
FUNCTION_BLOCK FB 1032
TITLE =A_3225_MXZ01MA FAN 1
//COPYRIGHT:     (C) 2009  BUHLER AG, CH-9240 UZWIL, SWITZERLAND
//
//PRODUCT:       WinCoS_BIW01_09
//
//TITLE:         FAN 1
//
//--------------------------------------------------------------------------------
//
//IDENT:         AUTHOR:             DEPT:                             DATE:
//
//P01_FB1032.1.0 K.Renz              CSB41                             09.Okt.2009
//               1st Release
//
//--------------------------------------------------------------------------------
//
//PURPOSE:
//
//MANUAL :
//
//RESTRICTIONS:
//
//--------------------------------------------------------------------------------
AUTHOR : KR
FAMILY : USW
VERSION : 0.0


VAR
  Ma : "GCS7_M_FB50_Data";	// Machine
  A_3225_KCU04 : "GCS7_E_DigInput";	// Mon1: DigInpCont
  A_3225_MXZ01_SM : "GCS7_E_DigInput";	// Mon2: DigInpCont
  Mon3 : "GCS7_E_DigInput";	// spare
  Mon4 : "GCS7_E_DigInput";	// spare
  Mon5 : "GCS7_E_DigInput";	// spare
  Mon6 : "GCS7_E_DigInput";	// spare
  A_3225_MXZ01 : "GCS7_E_Motor";	// Motor: Motor
END_VAR
BEGIN
NETWORK
TITLE =Call SSW

      UC    "GCS7_M_Motor6Mon";
END_FUNCTION_BLOCK


FUNCTION_BLOCK "G297M_Code"
TITLE =G297M FAN KILN 2
//COPYRIGHT:    (C) 2009  BUHLER AG, CH-9240 UZWIL, SWITZERLAND
//
//PRODUCT:      WinCoS_BIW01_09
//
//TITLE:        FAN KILN 2
//                Machine group control
//                Maschinengruppensteuerung
//
//--------------------------------------------------------------------------------
//
//IDENT:        AUTHOR:             DEPT:                              DATE:
//
//P01_FB397.1.0 K.Renz              CSB41                              09.Okt.2009
//             1st Release
//
//--------------------------------------------------------------------------------
//
//PURPOSE:
//
//MANUAL :
//
//RESTRICTIONS:
//
//--------------------------------------------------------------------------------
AUTHOR : KR
FAMILY : USW
VERSION : 9.9


VAR
  Gr : "GCS7_GrpCtrlSub";	//Standard interface to group
  InOutValue1 : DINT ;	//Data for user
  InOutValue2 : DINT ;	//Data for user
  OutWayConflict : BOOL ;	//Data for user
  OutSelectionOk : BOOL ;	//Data for user
  CmdNewValue : BOOL ;	//Data for user
  CmdNewJob : BOOL ;	//Data for user
  OutCodeOK : BOOL ;	//Data for user
  InEndOfJob : BOOL ;	//Data for user
  staWayOk : BOOL ;	//Data for user
  EdgeStartRelease : BOOL ;	//Data for user
  USW8 : BOOL ;	//Data for user
  USW9 : BOOL ;	//Data for user
  USW10 : BOOL ;	//Data for user
  USW11 : BOOL ;	//Data for user
  USW12 : BOOL ;	//Data for user
  USW13 : BOOL ;	//Data for user
  USW14 : BOOL ;	//Data for user
  USW15 : BOOL ;	//Data for user
  A_3225_KCU04AI1 : "GCS7_E_AnalogInput";	// AnaInp
  A_3225_KCU04AI2 : "GCS7_E_AnalogInput";	// AnaInp
  A_3225_BTE05 : "GCS7_E_AnalogInput";	// AnaInp
  A_3225_BTE06 : "GCS7_E_AnalogInput";	// AnaInp
  spare412 : ARRAY  [412 .. 445 ] OF BYTE ;
  A_3225_MXZ01MA : FB 1032;	// Motor+6DI
  A_3225_TSC01_AC : "GCS7_E_AnalogInput";	// AnaInp
  A_3225_TSC01_AF : "GCS7_E_AnalogInput";	// AnaInp
  A_3225_TSC01_AP : "GCS7_E_AnalogInput";	// AnaInp
  A_3225_TSC01_AT : "GCS7_E_AnalogInput";	// AnaInp
  A_3225_TSC01_COM : "SSA_SEW_MOVIDRIVE";	// FU_Siemens
  A_3226_KCU04AI1 : "GCS7_E_AnalogInput";	// AnaInp
  A_3226_KCU04AI2 : "GCS7_E_AnalogInput";	// AnaInp
  A_3226_BTE05 : "GCS7_E_AnalogInput";	// AnaInp
  A_3226_BTE06 : "GCS7_E_AnalogInput";	// AnaInp
  A_3226_MXZ01MA : FB 1033;	// Motor+6DI
  A_3226_TSC01_AC : "GCS7_E_AnalogInput";	// AnaInp
  A_3226_TSC01_AF : "GCS7_E_AnalogInput";	// AnaInp
  A_3226_TSC01_AP : "GCS7_E_AnalogInput";	// AnaInp
  A_3226_TSC01_AT : "GCS7_E_AnalogInput";	// AnaInp
  A_3226_TSC01_COM : "SSA_SEW_MOVIDRIVE";	// FU_Siemens
  A_3226_TSC01 : FB14;   // DigInpCont
END_VAR
VAR_TEMP
  tmpEnable : BOOL ;
  tmpFlag : BOOL ;
  tmpCmdNext : BOOL ;
  tmpLocal : BOOL ;
  tmpAspOk : BOOL ;
  tmpHWStop : BOOL ;
  tmpInstanzDBNo : INT ;
END_VAR
BEGIN
NETWORK
TITLE =



NETWORK
TITLE =Read command from group control
//Parameter
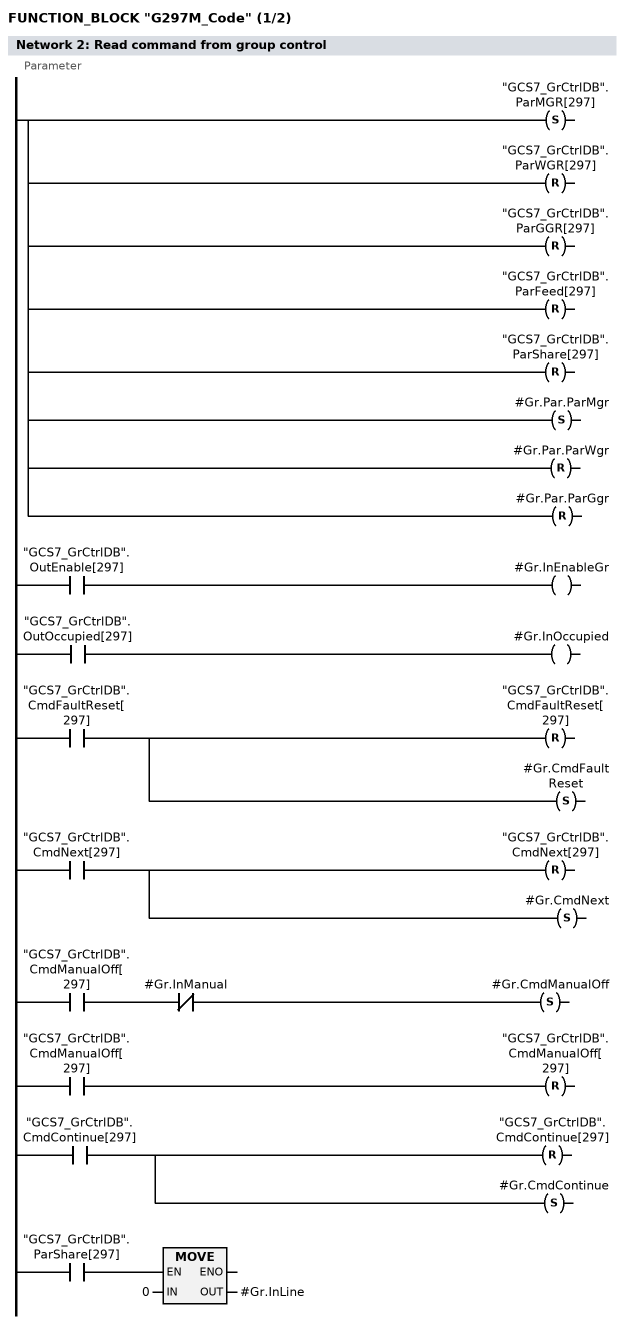
      SET   ;
      S     "GCS7_GrCtrlDB".ParMGR[297];
      R     "GCS7_GrCtrlDB".ParWGR[297];
      R     "GCS7_GrCtrlDB".ParGGR[297];
      R     "GCS7_GrCtrlDB".ParFeed[297];
      R     "GCS7_GrCtrlDB".ParShare[297];
      S     #Gr.Par.ParMgr;
      R     #Gr.Par.ParWgr;
      R     #Gr.Par.ParGgr;
//Command
      U     "GCS7_GrCtrlDB".OutEnable[297];
      =     #Gr.InEnableGr;
      U     "GCS7_GrCtrlDB".OutOccupied[297];
      =     #Gr.InOccupied;
      U     "GCS7_GrCtrlDB".CmdFaultReset[297];
      R     "GCS7_GrCtrlDB".CmdFaultReset[297];
      S     #Gr.CmdFaultReset;
      U     "GCS7_GrCtrlDB".CmdNext[297];
      R     "GCS7_GrCtrlDB".CmdNext[297];
      S     #Gr.CmdNext;

      U     "GCS7_GrCtrlDB".CmdManualOff[297];
      UN    #Gr.InManual;
      S     #Gr.CmdManualOff;
      U     "GCS7_GrCtrlDB".CmdManualOff[297];
      R     "GCS7_GrCtrlDB".CmdManualOff[297];

//      U     "GCS7_GrCtrlDB".CmdManualOff[297]
//      O     "GCS7_GrCtrlDB".OutOccupied[297]
//      R     "GCS7_GrCtrlDB".CmdManualOff[297]
//      S     #Gr.CmdManualOff

      U     "GCS7_GrCtrlDB".CmdContinue[297];
      R     "GCS7_GrCtrlDB".CmdContinue[297];
      S     #Gr.CmdContinue;
//Init Line Number
      U     "GCS7_GrCtrlDB".ParShare[297];
      SPBN  WE00;
      L     0;
      T     #Gr.InLine;
WE00: NOP   0;
NETWORK
TITLE =Call Methode Control
// 1. Handle Interface PCControl
// 2. Prepare mode --> ModePassive,ModeActive,ModeIdling
// 3. Reset global flags of the group
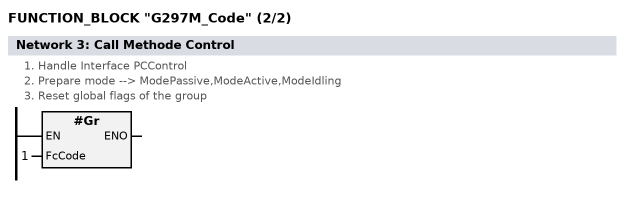
      CALL #Gr (
           FcCode                   := 1);
NETWORK
TITLE =Restart Idling Time

      L     #Gr.Par.ParIdling;
      L     2;
      >=I   ;
      SPB   IdTm;
      T     #Gr.Par.ParIdling;
IdTm: NOP   0;
      CLR   ;
      S     #Gr.CmdRestartIdling;
NETWORK
TITLE =Prepare global flags



NETWORK
TITLE =Set Pattern (Target position)

      U     #Gr.InManual;
      SPB   ILO6;

// Drehzahlabsenkung wenn die andere Horde im Cooling ist
// und die Temperatur unter der eigenen Horde 5°C > als T[Soll]
//      U     "MAL1S032Par".Par.FlagProcess.Cooling_Activ
//      U     "G302M".USW8                // Temperatur unter der Horde 5°C > T[Soll]
//      L     50                          // 50%
//      SPB   En06

      L     "MAL1S032Par".Par.ParIntProcess.SpeedVentilatorBasic;

//      U     "G275M".USW8                // Drehzahlverrinderung bei offenen Bypassklappen
//      SPBN  En06
//      L     DB799.DBW   26              // Sollwert vom LS
//      -I
//      SPA   En06
ILO6: NOP   0;
      L     "MAL1S033Par".Par.ParIntProcess.Speed_ILO_Fan;
      NOP   0;
      L     100;
      *I    ;
      T     #A_3225_TSC01_COM.OutValuePC; // xxx.xx%
      T     #A_3226_TSC01_COM.OutValuePC; // xxx.xx%


NETWORK
TITLE =Interlocking WayOk



NETWORK
TITLE =Interlocking Autostart

      CLR   ;
      R     #Gr.OutAutostart;
NETWORK
TITLE =Interlocking Enable
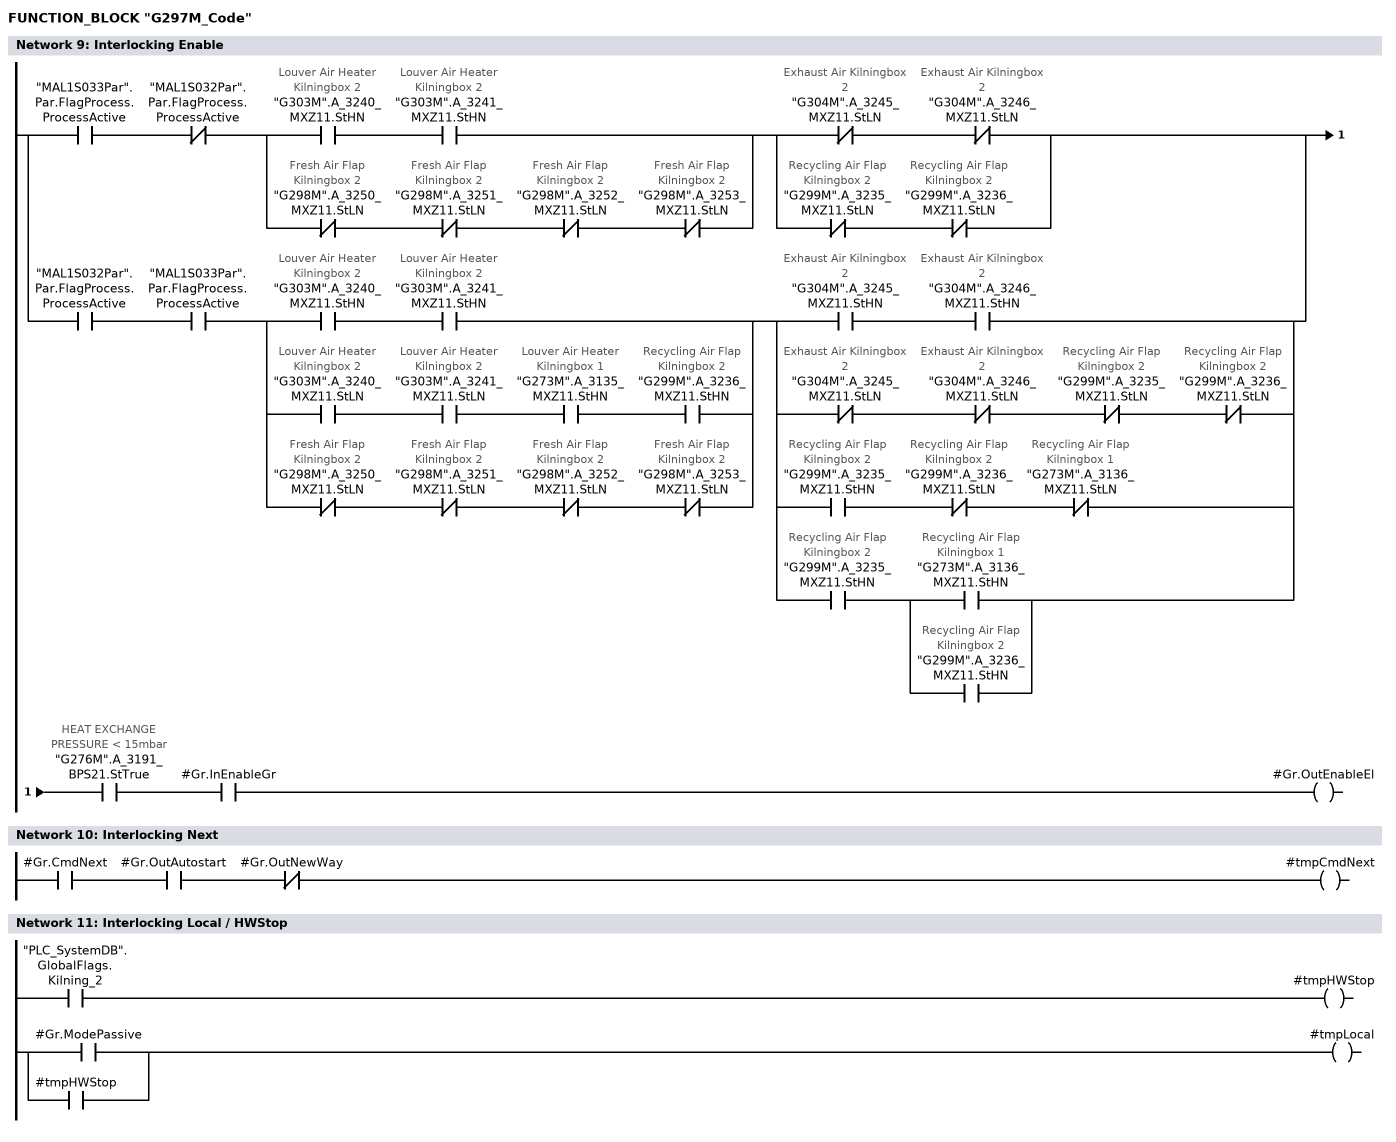

      U(    ;
//--------------------- Ein-Hordenbetrieb ----------------------------//
      U     "MAL1S033Par".Par.FlagProcess.ProcessActive;
      UN    "MAL1S032Par".Par.FlagProcess.ProcessActive;
// Luft-Eintritt
      U(    ;
      U     "G303M".A_3240_MXZ11.StHN; // Louver Air Heater Kilningbox 2
      U     "G303M".A_3241_MXZ11.StHN; // Louver Air Heater Kilningbox 2
      O     ;
      UN    "G298M".A_3250_MXZ11.StLN; // Fresh Air Flap Kilningbox 2
      UN    "G298M".A_3251_MXZ11.StLN; // Fresh Air Flap Kilningbox 2
      UN    "G298M".A_3252_MXZ11.StLN; // Fresh Air Flap Kilningbox 2
      UN    "G298M".A_3253_MXZ11.StLN; // Fresh Air Flap Kilningbox 2
      )     ;
// Luft-Austritt
      U(    ;
      UN    "G304M".A_3245_MXZ11.StLN; // Exhaust Air Kilningbox 2
      UN    "G304M".A_3246_MXZ11.StLN; // Exhaust Air Kilningbox 2
      O     ;
      UN    "G299M".A_3235_MXZ11.StLN; // Recycling Air Flap Kilningbox 2
      UN    "G299M".A_3236_MXZ11.StLN; // Recycling Air Flap Kilningbox 2
      )     ;
      O     ;
//---------------------- Zwei-Hordenbetrieb --------------------------//
      U     "MAL1S032Par".Par.FlagProcess.ProcessActive;
      U     "MAL1S033Par".Par.FlagProcess.ProcessActive;
// Luft-Eintritt
      U(    ;
      U     "G303M".A_3240_MXZ11.StHN; // Louver Air Heater Kilningbox 2
      U     "G303M".A_3241_MXZ11.StHN; // Louver Air Heater Kilningbox 2
      O     ;
      U     "G303M".A_3240_MXZ11.StLN; // Louver Air Heater Kilningbox 2
      U     "G303M".A_3241_MXZ11.StLN; // Louver Air Heater Kilningbox 2
      U     "G273M".A_3135_MXZ11.StHN; // Louver Air Heater Kilningbox 1
      U     "G299M".A_3236_MXZ11.StHN; // Recycling Air Flap Kilningbox 2
      O     ;
      UN    "G298M".A_3250_MXZ11.StLN; // Fresh Air Flap Kilningbox 2
      UN    "G298M".A_3251_MXZ11.StLN; // Fresh Air Flap Kilningbox 2
      UN    "G298M".A_3252_MXZ11.StLN; // Fresh Air Flap Kilningbox 2
      UN    "G298M".A_3253_MXZ11.StLN; // Fresh Air Flap Kilningbox 2
      )     ;
// Luft-Austritt
      U(    ;
      U     "G304M".A_3245_MXZ11.StHN; // Exhaust Air Kilningbox 2
      U     "G304M".A_3246_MXZ11.StHN; // Exhaust Air Kilningbox 2
      O     ;
      UN    "G304M".A_3245_MXZ11.StLN; // Exhaust Air Kilningbox 2
      UN    "G304M".A_3246_MXZ11.StLN; // Exhaust Air Kilningbox 2
      UN    "G299M".A_3235_MXZ11.StLN; // Recycling Air Flap Kilningbox 2
      UN    "G299M".A_3236_MXZ11.StLN; // Recycling Air Flap Kilningbox 2
      O     ;
      U     "G299M".A_3235_MXZ11.StHN; // Recycling Air Flap Kilningbox 2
      UN    "G299M".A_3236_MXZ11.StLN; // Recycling Air Flap Kilningbox 2
      UN    "G273M".A_3136_MXZ11.StLN; // Recycling Air Flap Kilningbox 1
      O     ;
// 100% Umluft-Betrieb
      U     "G299M".A_3235_MXZ11.StHN; // Recycling Air Flap Kilningbox 2
      U(    ;
      O     "G273M".A_3136_MXZ11.StHN; // Recycling Air Flap Kilningbox 1
      O     "G299M".A_3236_MXZ11.StHN; // Recycling Air Flap Kilningbox 2
      )     ;
      )     ;
      )     ;

      U     "G276M".A_3191_BPS21.StTrue; // HEAT EXCHANGE PRESSURE < 15mbar
      U     #Gr.InEnableGr;
      =     #Gr.OutEnableEl;

NETWORK
TITLE =Interlocking Next

      U     #Gr.CmdNext;
      U     #Gr.OutAutostart;
      UN    #Gr.OutNewWay;
      =     #tmpCmdNext;

NETWORK
TITLE =Interlocking Local / HWStop

      U     "PLC_SystemDB".GlobalFlags.Kilning_2;
      =     #tmpHWStop;

      U     #Gr.ModePassive;
      O     #tmpHWStop;
      =     #tmpLocal;

NETWORK
TITLE =Interlocking Start Warning

      NOP   0;
//- Restart after fault --
      U     #Gr.CmdFaultReset;
      U     #Gr.VarFault;
      S     "SYS_StartWarningDB".Area[11].CmdResetStartWarning;
//- Run Timer --
      AUF   "G297M";
      CALL "GCS7_StartWarning" , "SYS_StartWarningDB" (
           InModeHigher             := FALSE,
           InArea                   := 11,
           InEnable                 := #Gr.OutEnableEl,
           InLocal                  := #tmpLocal,
           InStarted                := #Gr.VarStarted,
           InCmdNext                := #tmpCmdNext,
           OutCmdNext               := #tmpCmdNext,
           OutStartwarning          := #Gr.VarStartwarning);
//- Store Startwarning done  --
//- Reset Autostart --
      U     "SYS_StartWarningDB".TmpArea.OutStartReleaseRunningL;
      FN    #EdgeStartRelease;
      U     #Gr.VarFault;
      R     #Gr.OutAutostart;
NETWORK
TITLE ==A-3225-KCU04AI1 : VIBRATION MONITOR FAN 1 CHANNEL 1
//Alarm Level = 10.00mm/sec
//Trip Level = 11.20mm/sec
      NOP   0;
//-InLocal---
      U     #tmpLocal;
      O     DB923.DBX 2509.0; // emergency regime without fan 1
      =     #A_3225_KCU04AI1.InLocal;
//
//-Monitoring---
      CLR   ;
      =     #A_3225_KCU04AI1.InMonLL;
      CLR   ;
      =     #A_3225_KCU04AI1.InMonL;
      CLR   ;
      =     #A_3225_KCU04AI1.InMonMid;
      CLR   ;
      =     #A_3225_KCU04AI1.InMonH;
      SET   ;
      =     #A_3225_KCU04AI1.InMonHH;
//
//-Read inputs---
      L     "A_3225_KCU04_AI1";
      L     0;
      <I    ;
      SPB   v003;
      TAK   ;
v003: T     #A_3225_KCU04AI1.InpValue;
      U     "PLC_SystemDB".GlobalFlags.Kilning_2;
      =     #A_3225_KCU04AI1.InHWStop;
      U     "PLC_DPInfo".Master[1].SlavesError[102];
      =     #A_3225_KCU04AI1.InDPFault;
//
//-Set Parameters---
// --> Erläuterung
      L     L#2540; // 20mA = 25.40mm/sec
      T     "G297M".A_3225_KCU04AI1.Par.ParUnitsByMaxDigit;
      L     L#10000; // OutValuePc=OutValueUnits
      T     "G297M".A_3225_KCU04AI1.Par.ParUnitsBy100Pc;
      L     L#-1; // -0.01mm/sec
      T     "G297M".A_3225_KCU04AI1.Par.ParLimitLL;
      L     L#0; // 0.00mm/sec
      T     "G297M".A_3225_KCU04AI1.Par.ParLimitL;
      L     L#1000; // 10.00mm/sec
      T     "G297M".A_3225_KCU04AI1.Par.ParLimitH;
      L     L#1120; // 11.20mm/sec
      T     "G297M".A_3225_KCU04AI1.Par.ParLimitHH;
      SET   ;
      =     "G297M".A_3225_KCU04AI1.Par.ParWarningLL;
      =     "G297M".A_3225_KCU04AI1.Par.ParWarningL;
      =     "G297M".A_3225_KCU04AI1.Par.ParWarningMid;
      =     "G297M".A_3225_KCU04AI1.Par.ParWarningH;
      =     "G297M".A_3225_KCU04AI1.Par.ParPreAlarmH;
      =     "G297M".A_3225_KCU04AI1.Par.ParPreAlarmHH;
      CLR   ;
      =     "G297M".A_3225_KCU04AI1.Par.ParWarningHH;
//
//-Call object control---
      CALL #A_3225_KCU04AI1 ;
//
//-Write outputs---
NETWORK
TITLE ==A-3225-KCU04AI2 : VIBRATION MONITOR FAN 1 CHANNEL 2
//Alarm Level = 10.00mm/sec
//Trip Level = 11.20mm/sec
      NOP   0;
//-InLocal---
      U     #tmpLocal;
      O     DB923.DBX 2509.0; // emergency regime without fan 1
      =     #A_3225_KCU04AI2.InLocal;
//
//-Monitoring---
      CLR   ;
      =     #A_3225_KCU04AI2.InMonLL;
      CLR   ;
      =     #A_3225_KCU04AI2.InMonL;
      CLR   ;
      =     #A_3225_KCU04AI2.InMonMid;
      CLR   ;
      =     #A_3225_KCU04AI2.InMonH;
      SET   ;
      =     #A_3225_KCU04AI2.InMonHH;
//
//-Read inputs---
      L     "A_3225_KCU04_AI2";
      L     0;
      <I    ;
      SPB   v004;
      TAK   ;
v004: T     #A_3225_KCU04AI2.InpValue;
      U     "PLC_SystemDB".GlobalFlags.Kilning_2;
      =     #A_3225_KCU04AI2.InHWStop;
      U     "PLC_DPInfo".Master[1].SlavesError[102];
      =     #A_3225_KCU04AI2.InDPFault;
//
//-Set Parameters---
// --> Erläuterung
      L     L#2540; // 20mA = 25.40mm/sec
      T     "G297M".A_3225_KCU04AI2.Par.ParUnitsByMaxDigit;
      L     L#10000; // OutValuePc=OutValueUnits
      T     "G297M".A_3225_KCU04AI2.Par.ParUnitsBy100Pc;
      L     L#-1; // -0.01mm/sec
      T     "G297M".A_3225_KCU04AI2.Par.ParLimitLL;
      L     L#0; // 0.00mm/sec
      T     "G297M".A_3225_KCU04AI2.Par.ParLimitL;
      L     L#1000; // 10.00mm/sec
      T     "G297M".A_3225_KCU04AI2.Par.ParLimitH;
      L     L#1120; // 11.20mm/sec
      T     "G297M".A_3225_KCU04AI2.Par.ParLimitHH;
      SET   ;
      =     "G297M".A_3225_KCU04AI2.Par.ParWarningLL;
      =     "G297M".A_3225_KCU04AI2.Par.ParWarningL;
      =     "G297M".A_3225_KCU04AI2.Par.ParWarningMid;
      =     "G297M".A_3225_KCU04AI2.Par.ParWarningH;
      =     "G297M".A_3225_KCU04AI2.Par.ParPreAlarmH;
      =     "G297M".A_3225_KCU04AI2.Par.ParPreAlarmHH;
      CLR   ;
      =     "G297M".A_3225_KCU04AI2.Par.ParWarningHH;
//
//-Call object control---
      CALL #A_3225_KCU04AI2 ;
//
//-Write outputs---
NETWORK
TITLE ==A-3225-BTE05 : TEMPERATURE BEARING TEMPERATUR SENSOR
//Alarm Level = 100.00°C
//Trip Level = 110.00°C
      NOP   0;
//-InLocal---
      U     #tmpLocal;
      O     DB923.DBX 2509.0; // emergency regime without fan 1
      =     #A_3225_BTE05.InLocal;
//
//-Monitoring---
      CLR   ;
      =     #A_3225_BTE05.InMonLL;
      CLR   ;
      =     #A_3225_BTE05.InMonL;
      CLR   ;
      =     #A_3225_BTE05.InMonMid;
      CLR   ;
      =     #A_3225_BTE05.InMonH;
      SET   ;
      =     #A_3225_BTE05.InMonHH;
//
//-Read inputs---
      L     "A_3225_BTE05_AI1";
      T     #A_3225_BTE05.InpValue;
      U     "PLC_SystemDB".GlobalFlags.Kilning_2;
      =     #A_3225_BTE05.InHWStop;
      U     "PLC_DPInfo".Master[1].SlavesError[102];
      =     #A_3225_BTE05.InDPFault;

//To Block Problems with Sensor
      L     600;
      T     "G297M".A_3225_BTE05.Par.ParMonTimeH;
      T     "G297M".A_3225_BTE05.Par.ParMonTimeHH;
//
//-Set Parameters---
// --> Erläuterung
      L     L#27648; // Temperature direkt
      T     "G297M".A_3225_BTE05.Par.ParUnitsByMaxDigit;
      L     L#10000; // OutValuePc=OutValueUnits
      T     "G297M".A_3225_BTE05.Par.ParUnitsBy100Pc;
      L     L#0; // 0.00°C
      T     "G297M".A_3225_BTE05.Par.ParLimitLL;
      L     L#100; // 1.00°C
      T     "G297M".A_3225_BTE05.Par.ParLimitL;
      L     L#10000; // 100.00°C
      T     "G297M".A_3225_BTE05.Par.ParLimitH;
      L     L#11000; // 110.00°C
      T     "G297M".A_3225_BTE05.Par.ParLimitHH;
      SET   ;
      =     "G297M".A_3225_BTE05.Par.ParWarningLL;
      =     "G297M".A_3225_BTE05.Par.ParWarningL;
      =     "G297M".A_3225_BTE05.Par.ParWarningMid;
      =     "G297M".A_3225_BTE05.Par.ParWarningH;
      =     "G297M".A_3225_BTE05.Par.ParPreAlarmH;
      =     "G297M".A_3225_BTE05.Par.ParPreAlarmHH;
      CLR   ;
      =     "G297M".A_3225_BTE05.Par.ParWarningHH;
//
//-Call object control---
      CALL #A_3225_BTE05 ;
//
//-Write outputs---
NETWORK
TITLE ==A-3225-BTE06 : TEMPERATURE BEARING TEMPERATUR SENSOR
//Alarm Level = 100.00°C
//Trip Level = 110.00°C
      NOP   0;
//-InLocal---
      U     #tmpLocal;
      O     DB923.DBX 2509.0; // emergency regime without fan 1
      =     #A_3225_BTE06.InLocal;
//
//-Monitoring---
      SET   ;
      =     #A_3225_BTE06.InMonLL;
      CLR   ;
      =     #A_3225_BTE06.InMonL;
      CLR   ;
      =     #A_3225_BTE06.InMonMid;
      CLR   ;
      =     #A_3225_BTE06.InMonH;
      SET   ;
      =     #A_3225_BTE06.InMonHH;
//
//-Read inputs---
      L     "A_3225_BTE06_AI1";
      T     #A_3225_BTE06.InpValue;
      U     "PLC_SystemDB".GlobalFlags.Kilning_2;
      =     #A_3225_BTE06.InHWStop;
      U     "PLC_DPInfo".Master[1].SlavesError[102];
      =     #A_3225_BTE06.InDPFault;

//To Block Problems with Sensor
      L     600;
      T     "G297M".A_3225_BTE06.Par.ParMonTimeH;
      T     "G297M".A_3225_BTE06.Par.ParMonTimeHH;
//
//-Set Parameters---
// --> Erläuterung
      L     L#27648; // Temperature direkt
      T     "G297M".A_3225_BTE06.Par.ParUnitsByMaxDigit;
      L     L#10000; // OutValuePc=OutValueUnits
      T     "G297M".A_3225_BTE06.Par.ParUnitsBy100Pc;
      L     L#0; // 0.00°C
      T     "G297M".A_3225_BTE06.Par.ParLimitLL;
      L     L#100; // 1.00°C
      T     "G297M".A_3225_BTE06.Par.ParLimitL;
      L     L#10000; // 100.00°C
      T     "G297M".A_3225_BTE06.Par.ParLimitH;
      L     L#11000; // 110.00°C
      T     "G297M".A_3225_BTE06.Par.ParLimitHH;
      SET   ;
      =     "G297M".A_3225_BTE06.Par.ParWarningLL;
      =     "G297M".A_3225_BTE06.Par.ParWarningL;
      =     "G297M".A_3225_BTE06.Par.ParWarningMid;
      =     "G297M".A_3225_BTE06.Par.ParWarningH;
      =     "G297M".A_3225_BTE06.Par.ParPreAlarmH;
      =     "G297M".A_3225_BTE06.Par.ParPreAlarmHH;
      CLR   ;
      =     "G297M".A_3225_BTE06.Par.ParWarningHH;
//
//-Call object control---
      CALL #A_3225_BTE06 ;
//
//-Write outputs---
NETWORK
TITLE ==A-3225-MXZ01MA : FAN 1
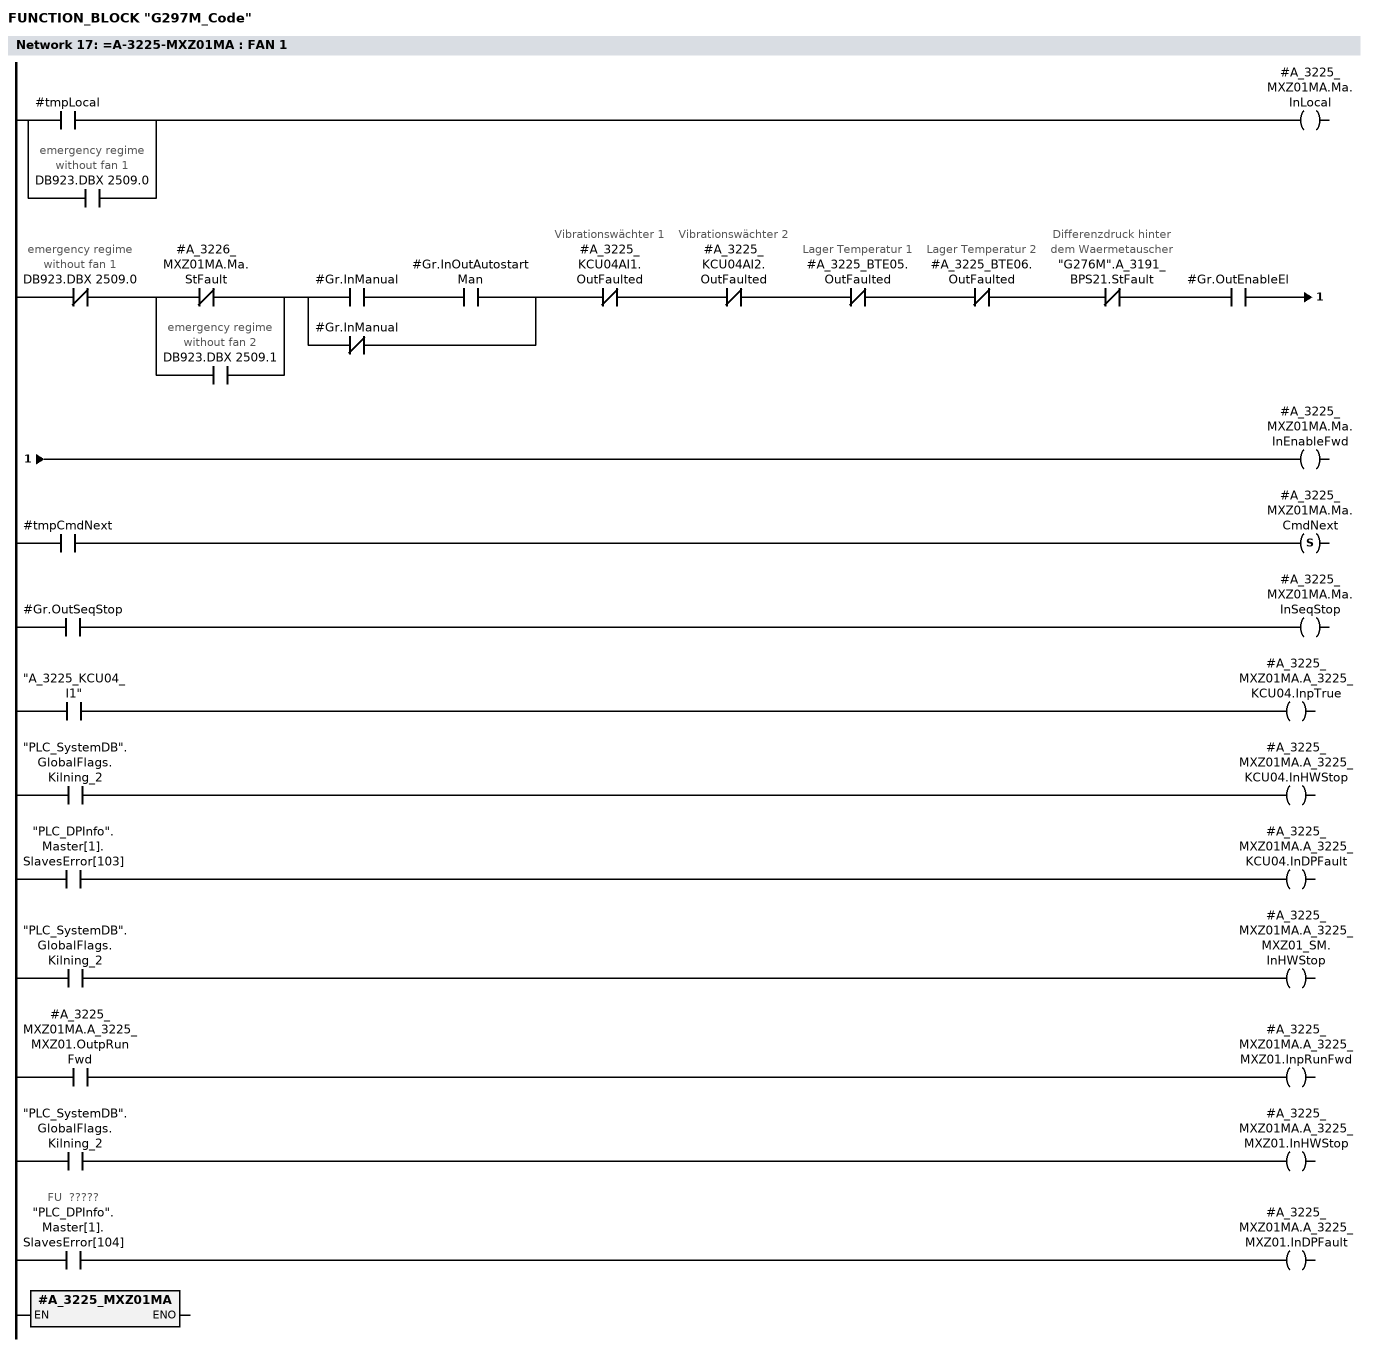

      NOP   0;
//-InLocal---
      U     #tmpLocal;
      O     DB923.DBX 2509.0; // emergency regime without fan 1
      =     #A_3225_MXZ01MA.Ma.InLocal;
//
//-Interlocking---
      UN    DB923.DBX 2509.0; // emergency regime without fan 1
      U(    ;
      UN    #A_3226_MXZ01MA.Ma.StFault;
      O     DB923.DBX 2509.1; // emergency regime without fan 2
      )     ;
      U(    ;
      U     #Gr.InManual;
      U     #Gr.InOutAutostartMan;
      ON    #Gr.InManual;
      )     ;
      UN    #A_3225_KCU04AI1.OutFaulted; // Vibrationswächter 1
      UN    #A_3225_KCU04AI2.OutFaulted; // Vibrationswächter 2
      UN    #A_3225_BTE05.OutFaulted; // Lager Temperatur 1
      UN    #A_3225_BTE06.OutFaulted; // Lager Temperatur 2
      UN    "G276M".A_3191_BPS21.StFault; // Differenzdruck hinter dem Waermetauscher
      U     #Gr.OutEnableEl;
      =     #A_3225_MXZ01MA.Ma.InEnableFwd;
//
      U     #tmpCmdNext;
//      U     "MAL1S033Par".Par.FlagProcess2.Schaltp_5
      S     #A_3225_MXZ01MA.Ma.CmdNext;
//
      U     #Gr.OutSeqStop;
      =     #A_3225_MXZ01MA.Ma.InSeqStop;
//
//=Values and commands of elements===
//-=A-3225-KCU04---
//      CLR
//      S     #A_3225_MXZ01MA.A_3225_KCU04.CmdRunTimeOutTime
//-=A-3225-MXZ01_SM---
//      CLR
//      S     #A_3225_MXZ01MA.A_3225_MXZ01_SM.CmdRunTimeOutTime
//
//-Read inputs of elements---
      U     "A_3225_KCU04_I1";
      =     #A_3225_MXZ01MA.A_3225_KCU04.InpTrue;
      U     "PLC_SystemDB".GlobalFlags.Kilning_2;
      =     #A_3225_MXZ01MA.A_3225_KCU04.InHWStop;
      U     "PLC_DPInfo".Master[1].SlavesError[103];
      =     #A_3225_MXZ01MA.A_3225_KCU04.InDPFault;
      U     "PLC_SystemDB".GlobalFlags.Kilning_2;
      =     #A_3225_MXZ01MA.A_3225_MXZ01_SM.InHWStop;
      U     #A_3225_MXZ01MA.A_3225_MXZ01.OutpRunFwd;
      =     #A_3225_MXZ01MA.A_3225_MXZ01.InpRunFwd;
      U     "PLC_SystemDB".GlobalFlags.Kilning_2;
      =     #A_3225_MXZ01MA.A_3225_MXZ01.InHWStop;

      U     "PLC_DPInfo".Master[1].SlavesError[104]; // FU  ?????
      =     #A_3225_MXZ01MA.A_3225_MXZ01.InDPFault;
//
//-Set Parameters---
//
//-Call object control---
      CALL #A_3225_MXZ01MA ;
//
//-Write outputs---
NETWORK
TITLE ==A-3225-TSC01_COM : FAN 1 FU KOMMUNIKATION

      NOP   0;
      U     #A_3225_MXZ01MA.A_3225_MXZ01.OutpRunFwd;
      =     #A_3225_TSC01_COM.InEnableFwd;
//      U     #A_3225_MXZ01MA.A_3225_MXZ01.OutpRunRev
      CLR   ;
      =     #A_3225_TSC01_COM.InEnableRev;
      U     #Gr.CmdFaultReset;
      O     #A_3225_MXZ01MA.A_3225_KCU04.OutpFaultReset;
      S     #A_3225_TSC01_COM.CmdFaultReset;

//
//-Read inputs---
//
//-Set Parameters---
      U     "PLC_SystemDB".GlobalFlags.StaTest;
      SPB   NCo1;
//
//-Call object control---
      CALL #A_3225_TSC01_COM ;
//
//-Write outputs---
NCo1: NOP   0;
// Simu
      U     "PLC_SystemDB".GlobalFlags.StaTest;
      U     #A_3225_MXZ01MA.A_3225_MXZ01.StStartedFwd;
      SPBN  ACT1;
      L     #A_3225_TSC01_COM.Output.SetpointValue01; // xxx.xx%
      L     6;
      /I    ;
      L     10;
      *I    ;
      T     #A_3225_TSC01_COM.Input.ActualValue01;

      L     675; // 675A
      T     #A_3225_TSC01_COM.Input.ActualValue02;
ACT1: NOP   0;
NETWORK
TITLE ==A-3225-TSC01_AC : ACT. CURRENT FAN 1 FU

      NOP   0;
//-InLocal---
      U     #tmpLocal;
      O     DB923.DBX 2509.0; // emergency regime without fan 1
      =     #A_3225_TSC01_AC.InLocal;
//
//-Monitoring---
      CLR   ;
      =     #A_3225_TSC01_AC.InMonLL;
      CLR   ;
      =     #A_3225_TSC01_AC.InMonL;
      CLR   ;
      =     #A_3225_TSC01_AC.InMonMid;
      CLR   ;
      =     #A_3225_TSC01_AC.InMonH;
      CLR   ;
      =     #A_3225_TSC01_AC.InMonHH;
//
//-Read inputs---
      L     #A_3225_TSC01_COM.Output.SetpointValue02;
      T     #A_3225_TSC01_AC.InpValue;
      U     "PLC_SystemDB".GlobalFlags.Kilning_2;
      =     #A_3225_TSC01_AC.InHWStop;
//
//-Set Parameters---
// --> Erläuterung
      L     L#9113; // Stromwert bei 27648Dez
      T     "G297M".A_3225_TSC01_AC.Par.ParUnitsByMaxDigit;
      L     L#10000; // OutValuePc=OutValueUnits
      T     "G297M".A_3225_TSC01_AC.Par.ParUnitsBy100Pc;
      L     L#0; // 0.0A
      T     "G297M".A_3225_TSC01_AC.Par.ParLimitLL;
      L     L#4000; // 40.0A
      T     "G297M".A_3225_TSC01_AC.Par.ParLimitL;
      L     L#5400; // 540.0A=100.0%
      T     "G297M".A_3225_TSC01_AC.Par.ParLimitH;
      L     L#7000; // 700.0A=130.0%
      T     "G297M".A_3225_TSC01_AC.Par.ParLimitHH;
//
//-Call object control---
      CALL #A_3225_TSC01_AC ;
//
//-Write outputs---
NETWORK
TITLE ==A-3225-TSC01_AF : ACT. FREQUENCY FAN 1 FU

      NOP   0;
//-InLocal---
      U     #tmpLocal;
      O     DB923.DBX 2509.0; // emergency regime without fan 1
      =     #A_3225_TSC01_AF.InLocal;
//
//-Monitoring---
      CLR   ;
      =     #A_3225_TSC01_AF.InMonLL;
      CLR   ;
      =     #A_3225_TSC01_AF.InMonL;
      CLR   ;
      =     #A_3225_TSC01_AF.InMonMid;
      CLR   ;
      =     #A_3225_TSC01_AF.InMonH;
      CLR   ;
      =     #A_3225_TSC01_AF.InMonHH;
//
//-Read inputs---
      L     #A_3225_TSC01_COM.InValuePC; // Umgerechnet in FU-FB
      T     #A_3225_TSC01_AF.InpValue;
      U     "PLC_SystemDB".GlobalFlags.Kilning_2;
      =     #A_3225_TSC01_AF.InHWStop;
//
//-Set Parameters---
// --> Erläuterung
      L     L#27648; // InpValue=Drehzahl direkt
      T     "G297M".A_3225_TSC01_AF.Par.ParUnitsByMaxDigit;
      L     L#10000; // OutValuePc=OutValueUnits
      T     "G297M".A_3225_TSC01_AF.Par.ParUnitsBy100Pc;
      L     L#4000; // 40.00% ist untere Grenze
      T     "G297M".A_3225_TSC01_AF.Par.ParLimitLL;
      L     L#4100; // 41.00%
      T     "G297M".A_3225_TSC01_AF.Par.ParLimitL;
      L     L#8000; // 80.00%
      T     "G297M".A_3225_TSC01_AF.Par.ParLimitH;
      L     L#10100; // 101.00%
      T     "G297M".A_3225_TSC01_AF.Par.ParLimitHH;
//
//-Call object control---
      CALL #A_3225_TSC01_AF ;
//
//-Write outputs---
NETWORK
TITLE ==A-3225-TSC01_AP : ACT. POWER FAN 1 FU

      NOP   0;
//-InLocal---
      U     #tmpLocal;
      O     DB923.DBX 2509.0; // emergency regime without fan 1
      =     #A_3225_TSC01_AP.InLocal;
//
//-Monitoring---
      CLR   ;
      =     #A_3225_TSC01_AP.InMonLL;
      CLR   ;
      =     #A_3225_TSC01_AP.InMonL;
      CLR   ;
      =     #A_3225_TSC01_AP.InMonMid;
      CLR   ;
      =     #A_3225_TSC01_AP.InMonH;
      CLR   ;
      =     #A_3225_TSC01_AP.InMonHH;
//
//-Read inputs---
      L     #A_3225_TSC01_COM.Output.SetpointValue03;
      T     #A_3225_TSC01_AP.InpValue;
      U     "PLC_SystemDB".GlobalFlags.Kilning_2;
      =     #A_3225_TSC01_AP.InHWStop;
//
//-Set Parameters---
// --> Erläuterung
      L     L#10650; // Leistung bei 27648Dez
      T     "G297M".A_3225_TSC01_AP.Par.ParUnitsByMaxDigit;
      L     L#10000; // OutValuePc=OutValueUnits
      T     "G297M".A_3225_TSC01_AP.Par.ParUnitsBy100Pc;
      L     L#0; // 0.0kW
      T     "G297M".A_3225_TSC01_AP.Par.ParLimitLL;
      L     L#100; // 10.0kW
      T     "G297M".A_3225_TSC01_AP.Par.ParLimitL;
      L     L#3150; // 315.0kW Motorleistung
      T     "G297M".A_3225_TSC01_AP.Par.ParLimitH;
      L     L#7000; // 631.1kW Leistung FU
      T     "G297M".A_3225_TSC01_AP.Par.ParLimitHH;
//
//-Call object control---
      CALL #A_3225_TSC01_AP ;
//
//-Write outputs---
NETWORK
TITLE ==A-3225-TSC01_AT : ACT. TORQUE FAN 1 FU

      NOP   0;
//-InLocal---
      U     #tmpLocal;
      O     DB923.DBX 2509.0; // emergency regime without fan 1
      =     #A_3225_TSC01_AT.InLocal;
//
//-Monitoring---
      CLR   ;
      =     #A_3225_TSC01_AT.InMonLL;
      CLR   ;
      =     #A_3225_TSC01_AT.InMonL;
      CLR   ;
      =     #A_3225_TSC01_AT.InMonMid;
      CLR   ;
      =     #A_3225_TSC01_AT.InMonH;
      CLR   ;
      =     #A_3225_TSC01_AT.InMonHH;
//
//-Read inputs---
      L     #A_3225_TSC01_COM.Output.SetpointValue04;
      L     0;
      U     #A_3225_TSC01_COM.Input.StateWord_1.BETRIEBSBEREIT;
      SPBN  M220;
      L     1500;
M220: T     #A_3225_TSC01_AT.InpValue;
      U     "PLC_SystemDB".GlobalFlags.Kilning_2;
      =     #A_3225_TSC01_AT.InHWStop;
//
//-Set Parameters---
// --> Erläuterung
      L     L#6835; // Drehmoment bei 27648Dez
      T     "G297M".A_3225_TSC01_AT.Par.ParUnitsByMaxDigit;
      L     L#10000; // OutValuePc=OutValueUnits
      T     "G297M".A_3225_TSC01_AT.Par.ParUnitsBy100Pc;
      L     L#0; // 0Nm
      T     "G297M".A_3225_TSC01_AT.Par.ParLimitLL;
      L     L#10; // 10Nm
      T     "G297M".A_3225_TSC01_AT.Par.ParLimitL;
      L     L#4050; // 4050Nm
      T     "G297M".A_3225_TSC01_AT.Par.ParLimitH;
      L     L#6835; // 6835Nm
      T     "G297M".A_3225_TSC01_AT.Par.ParLimitHH;
//
//-Call object control---
      CALL #A_3225_TSC01_AT ;
//
//-Write outputs---
NETWORK
TITLE ==A-3226-KCU04AI1 : VIBRATION MONITOR FAN 2 CHANNEL 1
//Alarm Level = 10.00mm/sec
//Trip Level = 11.20mm/sec
      NOP   0;
//-InLocal---
      U     #tmpLocal;
      O     DB923.DBX 2509.1; // emergency regime without fan 2
      =     #A_3226_KCU04AI1.InLocal;
//
//-Monitoring---
      CLR   ;
      =     #A_3226_KCU04AI1.InMonLL;
      CLR   ;
      =     #A_3226_KCU04AI1.InMonL;
      CLR   ;
      =     #A_3226_KCU04AI1.InMonMid;
      SET   ;
      =     #A_3226_KCU04AI1.InMonH;
      SET   ;
      =     #A_3226_KCU04AI1.InMonHH;
//
//-Read inputs---
      L     "A_3226_KCU04_AI1";
      L     0;
      <I    ;
      SPB   v013;
      TAK   ;
v013: T     #A_3226_KCU04AI1.InpValue;
      U     "PLC_SystemDB".GlobalFlags.Kilning_2;
      =     #A_3226_KCU04AI1.InHWStop;
      U     "PLC_DPInfo".Master[1].SlavesError[102];
      =     #A_3226_KCU04AI1.InDPFault;
//
//-Set Parameters---
// --> Erläuterung
      L     L#2540; // 20mA = 25.40mm/sec
      T     "G297M".A_3226_KCU04AI1.Par.ParUnitsByMaxDigit;
      L     L#10000; // OutValuePc=OutValueUnits
      T     "G297M".A_3226_KCU04AI1.Par.ParUnitsBy100Pc;
      L     L#-1; // -0.01mm/sec
      T     "G297M".A_3226_KCU04AI1.Par.ParLimitLL;
      L     L#0; // 0.00mm/sec
      T     "G297M".A_3226_KCU04AI1.Par.ParLimitL;
      L     L#1000; // 10.00mm/sec
      T     "G297M".A_3226_KCU04AI1.Par.ParLimitH;
      L     L#1120; // 11.20mm/sec
      T     "G297M".A_3226_KCU04AI1.Par.ParLimitHH;
      SET   ;
      =     "G297M".A_3226_KCU04AI1.Par.ParWarningLL;
      =     "G297M".A_3226_KCU04AI1.Par.ParWarningL;
      =     "G297M".A_3226_KCU04AI1.Par.ParWarningMid;
      =     "G297M".A_3226_KCU04AI1.Par.ParWarningH;
      =     "G297M".A_3226_KCU04AI1.Par.ParPreAlarmH;
      =     "G297M".A_3226_KCU04AI1.Par.ParPreAlarmHH;
      CLR   ;
      =     "G297M".A_3226_KCU04AI1.Par.ParWarningHH;
//
//-Call object control---
      CALL #A_3226_KCU04AI1 ;
//
//-Write outputs---
NETWORK
TITLE ==A-3226-KCU04AI2 : VIBRATION MONITOR FAN 2 CHANNEL 2
//Alarm Level = 10.00mm/sec
//Trip Level = 11.20mm/sec
      NOP   0;
//-InLocal---
      U     #tmpLocal;
      O     DB923.DBX 2509.1; // emergency regime without fan 2
      =     #A_3226_KCU04AI2.InLocal;
//
//-Monitoring---
      CLR   ;
      =     #A_3226_KCU04AI2.InMonLL;
      CLR   ;
      =     #A_3226_KCU04AI2.InMonL;
      CLR   ;
      =     #A_3226_KCU04AI2.InMonMid;
      SET   ;
      =     #A_3226_KCU04AI2.InMonH;
      SET   ;
      =     #A_3226_KCU04AI2.InMonHH;
//
//-Read inputs---
      L     "A_3226_KCU04_AI2";
      L     0;
      <I    ;
      SPB   v014;
      TAK   ;
v014: T     #A_3226_KCU04AI2.InpValue;
      U     "PLC_SystemDB".GlobalFlags.Kilning_2;
      =     #A_3226_KCU04AI2.InHWStop;
      U     "PLC_DPInfo".Master[1].SlavesError[102];
      =     #A_3226_KCU04AI2.InDPFault;
//
//-Set Parameters---
// --> Erläuterung
      L     L#2540; // 20mA = 25.40mm/sec
      T     "G297M".A_3226_KCU04AI2.Par.ParUnitsByMaxDigit;
      L     L#10000; // OutValuePc=OutValueUnits
      T     "G297M".A_3226_KCU04AI2.Par.ParUnitsBy100Pc;
      L     L#-1; // -0.01mm/sec
      T     "G297M".A_3226_KCU04AI2.Par.ParLimitLL;
      L     L#0; // 0.00mm/sec
      T     "G297M".A_3226_KCU04AI2.Par.ParLimitL;
      L     L#1000; // 10.00mm/sec
      T     "G297M".A_3226_KCU04AI2.Par.ParLimitH;
      L     L#1120; // 11.20mm/sec
      T     "G297M".A_3226_KCU04AI2.Par.ParLimitHH;
      SET   ;
      =     "G297M".A_3226_KCU04AI2.Par.ParWarningLL;
      =     "G297M".A_3226_KCU04AI2.Par.ParWarningL;
      =     "G297M".A_3226_KCU04AI2.Par.ParWarningMid;
      =     "G297M".A_3226_KCU04AI2.Par.ParWarningH;
      =     "G297M".A_3226_KCU04AI2.Par.ParPreAlarmH;
      =     "G297M".A_3226_KCU04AI2.Par.ParPreAlarmHH;
      CLR   ;
      =     "G297M".A_3226_KCU04AI2.Par.ParWarningHH;
//
//-Call object control---
      CALL #A_3226_KCU04AI2 ;
//
//-Write outputs---
NETWORK
TITLE ==A-3226-BTE05 : TEMPERATURE BEARING TEMPERATUR SENSOR
//Alarm Level = 100.00°C
//Trip Level = 110.00°C
      NOP   0;
//-InLocal---
      U     #tmpLocal;
      O     DB923.DBX 2509.1; // emergency regime without fan 2
      =     #A_3226_BTE05.InLocal;
//
//-Monitoring---
      CLR   ;
      =     #A_3226_BTE05.InMonLL;
      CLR   ;
      =     #A_3226_BTE05.InMonL;
      CLR   ;
      =     #A_3226_BTE05.InMonMid;
      SET   ;
      =     #A_3226_BTE05.InMonH;
      SET   ;
      =     #A_3226_BTE05.InMonHH;
//
//-Read inputs---
      L     "A_3226_BTE05_AI1";
      T     #A_3226_BTE05.InpValue;
      U     "PLC_SystemDB".GlobalFlags.Kilning_2;
      =     #A_3226_BTE05.InHWStop;
      U     "PLC_DPInfo".Master[1].SlavesError[102];
      =     #A_3226_BTE05.InDPFault;

//To Block Problems with Sensor
      L     600;
      T     "G297M".A_3226_BTE05.Par.ParMonTimeH;
      T     "G297M".A_3226_BTE05.Par.ParMonTimeHH;
//
//-Set Parameters---
// --> Erläuterung
      L     L#27648; // Temperature direkt
      T     "G297M".A_3226_BTE05.Par.ParUnitsByMaxDigit;
      L     L#10000; // OutValuePc=OutValueUnits
      T     "G297M".A_3226_BTE05.Par.ParUnitsBy100Pc;
      L     L#0; // 0.00°C
      T     "G297M".A_3226_BTE05.Par.ParLimitLL;
      L     L#100; // 1.00°C
      T     "G297M".A_3226_BTE05.Par.ParLimitL;
      L     L#10000; // 100.00°C
      T     "G297M".A_3226_BTE05.Par.ParLimitH;
      L     L#11000; // 110.00°C
      T     "G297M".A_3226_BTE05.Par.ParLimitHH;
      SET   ;
      =     "G297M".A_3226_BTE05.Par.ParWarningLL;
      =     "G297M".A_3226_BTE05.Par.ParWarningL;
      =     "G297M".A_3226_BTE05.Par.ParWarningMid;
      =     "G297M".A_3226_BTE05.Par.ParWarningH;
      =     "G297M".A_3226_BTE05.Par.ParPreAlarmH;
      =     "G297M".A_3226_BTE05.Par.ParPreAlarmHH;
      CLR   ;
      =     "G297M".A_3226_BTE05.Par.ParWarningHH;
//
//-Call object control---
      CALL #A_3226_BTE05 ;
//
//-Write outputs---
NETWORK
TITLE ==A-3226-BTE06 : TEMPERATURE BEARING TEMPERATUR SENSOR
//Alarm Level = 100.00°C
//Trip Level = 110.00°C
      NOP   0;
//-InLocal---
      U     #tmpLocal;
      O     DB923.DBX 2509.1; // emergency regime without fan 2
      =     #A_3226_BTE06.InLocal;
//
//-Monitoring---
      CLR   ;
      =     #A_3226_BTE06.InMonLL;
      CLR   ;
      =     #A_3226_BTE06.InMonL;
      CLR   ;
      =     #A_3226_BTE06.InMonMid;
      SET   ;
      =     #A_3226_BTE06.InMonH;
      SET   ;
      =     #A_3226_BTE06.InMonHH;
//
//-Read inputs---
      L     "A_3226_BTE06_AI1";
      T     #A_3226_BTE06.InpValue;
      U     "PLC_SystemDB".GlobalFlags.Kilning_2;
      =     #A_3226_BTE06.InHWStop;
      U     "PLC_DPInfo".Master[1].SlavesError[102];
      =     #A_3226_BTE06.InDPFault;

//To Block Problems with Sensor
      L     600;
      T     "G297M".A_3226_BTE06.Par.ParMonTimeH;
      T     "G297M".A_3226_BTE06.Par.ParMonTimeHH;
//
//-Set Parameters---
// --> Erläuterung
      L     L#27648; // Temperature direkt
      T     "G297M".A_3226_BTE06.Par.ParUnitsByMaxDigit;
      L     L#10000; // OutValuePc=OutValueUnits
      T     "G297M".A_3226_BTE06.Par.ParUnitsBy100Pc;
      L     L#0; // 0.00°C
      T     "G297M".A_3226_BTE06.Par.ParLimitLL;
      L     L#100; // 1.00°C
      T     "G297M".A_3226_BTE06.Par.ParLimitL;
      L     L#10000; // 100.00°C
      T     "G297M".A_3226_BTE06.Par.ParLimitH;
      L     L#11000; // 110.00°C
      T     "G297M".A_3226_BTE06.Par.ParLimitHH;
      SET   ;
      =     "G297M".A_3226_BTE06.Par.ParWarningLL;
      =     "G297M".A_3226_BTE06.Par.ParWarningL;
      =     "G297M".A_3226_BTE06.Par.ParWarningMid;
      =     "G297M".A_3226_BTE06.Par.ParWarningH;
      =     "G297M".A_3226_BTE06.Par.ParPreAlarmH;
      =     "G297M".A_3226_BTE06.Par.ParPreAlarmHH;
      CLR   ;
      =     "G297M".A_3226_BTE06.Par.ParWarningHH;
//
//-Call object control---
      CALL #A_3226_BTE06 ;
//
//-Write outputs---
NETWORK
TITLE ==A-3226-MXZ01MA : FAN 2
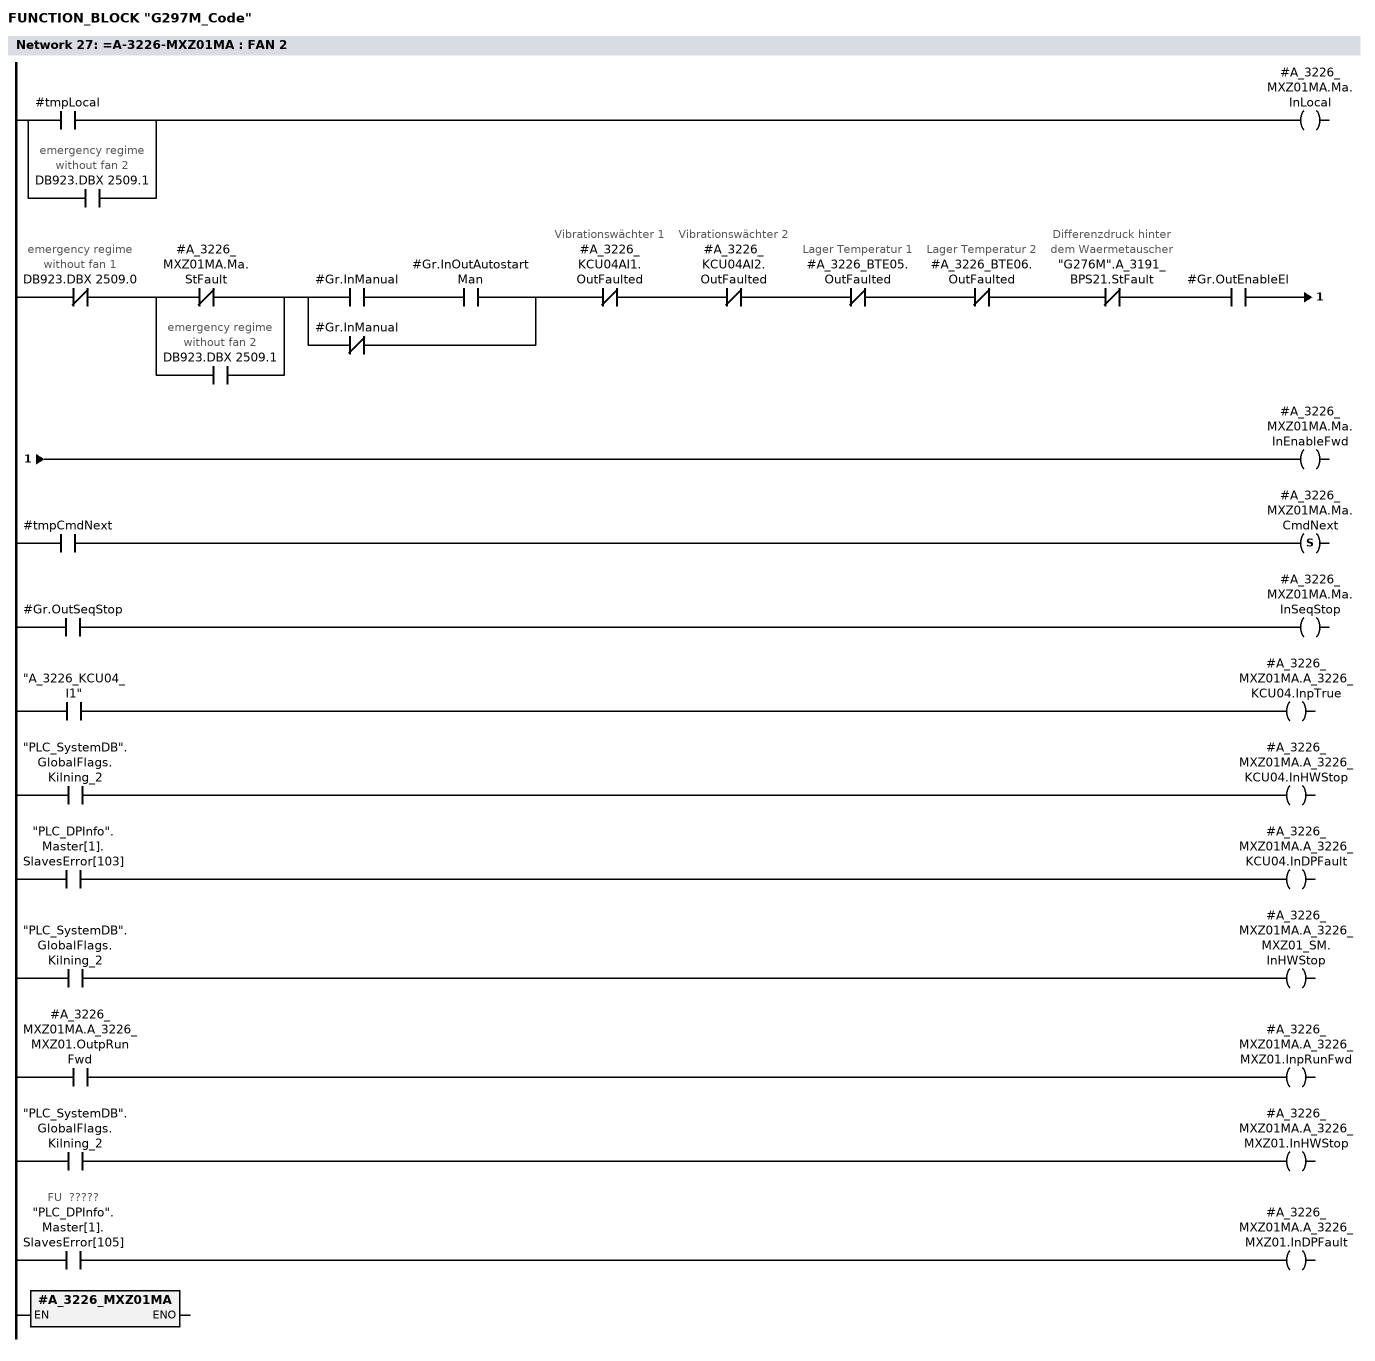

      NOP   0;
//-InLocal---
      U     #tmpLocal;
      O     DB923.DBX 2509.1; // emergency regime without fan 2
      =     #A_3226_MXZ01MA.Ma.InLocal;
//
//-Interlocking---
      UN    DB923.DBX 2509.0; // emergency regime without fan 1
      U(    ;
      UN    #A_3226_MXZ01MA.Ma.StFault;
      O     DB923.DBX 2509.1; // emergency regime without fan 2
      )     ;
      U(    ;
      U     #Gr.InManual;
      U     #Gr.InOutAutostartMan;
      ON    #Gr.InManual;
      )     ;
      UN    #A_3226_KCU04AI1.OutFaulted; // Vibrationswächter 1
      UN    #A_3226_KCU04AI2.OutFaulted; // Vibrationswächter 2
      UN    #A_3226_BTE05.OutFaulted; // Lager Temperatur 1
      UN    #A_3226_BTE06.OutFaulted; // Lager Temperatur 2
      UN    "G276M".A_3191_BPS21.StFault; // Differenzdruck hinter dem Waermetauscher
      U     #Gr.OutEnableEl;
      =     #A_3226_MXZ01MA.Ma.InEnableFwd;
//
      U     #tmpCmdNext;
//      U     "MAL1S033Par".Par.FlagProcess2.Schaltp_5
      S     #A_3226_MXZ01MA.Ma.CmdNext;
//
      U     #Gr.OutSeqStop;
      =     #A_3226_MXZ01MA.Ma.InSeqStop;
//
//=Values and commands of elements===
//-=A-3226-KCU04---
//      CLR
//      S     #A_3226_MXZ01MA.A_3226_KCU04.CmdRunTimeOutTime
//-=A-3226-MXZ01_SM---
//      CLR
//      S     #A_3226_MXZ01MA.A_3226_MXZ01_SM.CmdRunTimeOutTime
//
//-Read inputs of elements---
      U     "A_3226_KCU04_I1";
      =     #A_3226_MXZ01MA.A_3226_KCU04.InpTrue;
      U     "PLC_SystemDB".GlobalFlags.Kilning_2;
      =     #A_3226_MXZ01MA.A_3226_KCU04.InHWStop;
      U     "PLC_DPInfo".Master[1].SlavesError[103];
      =     #A_3226_MXZ01MA.A_3226_KCU04.InDPFault;
      U     "PLC_SystemDB".GlobalFlags.Kilning_2;
      =     #A_3226_MXZ01MA.A_3226_MXZ01_SM.InHWStop;
      U     #A_3226_MXZ01MA.A_3226_MXZ01.OutpRunFwd;
      =     #A_3226_MXZ01MA.A_3226_MXZ01.InpRunFwd;
      U     "PLC_SystemDB".GlobalFlags.Kilning_2;
      =     #A_3226_MXZ01MA.A_3226_MXZ01.InHWStop;

      U     "PLC_DPInfo".Master[1].SlavesError[105]; // FU  ?????
      =     #A_3226_MXZ01MA.A_3226_MXZ01.InDPFault;
//
//-Set Parameters---
//
//-Call object control---
      CALL #A_3226_MXZ01MA ;
//
//-Write outputs---
NETWORK
TITLE ==A-3226-TSC01_COM : FAN 2 FU KOMMUNIKATION

      NOP   0;
      U     #A_3226_MXZ01MA.A_3226_MXZ01.OutpRunFwd;
      =     #A_3226_TSC01_COM.InEnableFwd;
//      U     #A_3226_MXZ01MA.A_3226_MXZ01.OutpRunRev
      CLR   ;
      =     #A_3226_TSC01_COM.InEnableRev;
      U     #Gr.CmdFaultReset;
      O     #A_3226_MXZ01MA.A_3226_KCU04.OutpFaultReset;
      S     #A_3226_TSC01_COM.CmdFaultReset;

//
//-Read inputs---
//
//-Set Parameters---
      U     "PLC_SystemDB".GlobalFlags.StaTest;
      SPB   NCo2;
//
//-Call object control---
      CALL #A_3226_TSC01_COM ;
//
//-Write outputs---
NCo2: NOP   0;
// Simu
      U     "PLC_SystemDB".GlobalFlags.StaTest;
      U     #A_3226_MXZ01MA.A_3226_MXZ01.StStartedFwd;
      SPBN  ACT2;
      L     #A_3226_TSC01_COM.Output.SetpointValue01; // xxx.xx%
      L     6;
      /I    ;
      L     10;
      *I    ;
      T     #A_3226_TSC01_COM.Input.ActualValue01;

      L     675; // 675A
      T     #A_3226_TSC01_COM.Input.ActualValue02;
ACT2: NOP   0;
NETWORK
TITLE ==A-3226-TSC01_AC : ACT. CURRENT FAN 2 FU

      NOP   0;
//-InLocal---
      U     #tmpLocal;
      O     DB923.DBX 2509.1; // emergency regime without fan 2
      =     #A_3226_TSC01_AC.InLocal;
//
//-Monitoring---
      CLR   ;
      =     #A_3226_TSC01_AC.InMonLL;
      CLR   ;
      =     #A_3226_TSC01_AC.InMonL;
      CLR   ;
      =     #A_3226_TSC01_AC.InMonMid;
      CLR   ;
      =     #A_3226_TSC01_AC.InMonH;
      CLR   ;
      =     #A_3226_TSC01_AC.InMonHH;
//
//-Read inputs---
      L     #A_3226_TSC01_COM.Output.SetpointValue02;
      T     #A_3226_TSC01_AC.InpValue;
      U     "PLC_SystemDB".GlobalFlags.Kilning_2;
      =     #A_3226_TSC01_AC.InHWStop;
//
//-Set Parameters---
// --> Erläuterung
      L     L#9113; // Stromwert bei 27648Dez
      T     "G297M".A_3226_TSC01_AC.Par.ParUnitsByMaxDigit;
      L     L#10000; // OutValuePc=OutValueUnits
      T     "G297M".A_3226_TSC01_AC.Par.ParUnitsBy100Pc;
      L     L#0; // 0.0A
      T     "G297M".A_3226_TSC01_AC.Par.ParLimitLL;
      L     L#4000; // 40.0A
      T     "G297M".A_3226_TSC01_AC.Par.ParLimitL;
      L     L#5400; // 540.0A=100.0%
      T     "G297M".A_3226_TSC01_AC.Par.ParLimitH;
      L     L#7000; // 700.0A=130.0%
      T     "G297M".A_3226_TSC01_AC.Par.ParLimitHH;
//
//-Call object control---
      CALL #A_3226_TSC01_AC ;
//
//-Write outputs---
NETWORK
TITLE ==A-3226-TSC01_AF : ACT. FREQUENCY FAN 2 FU

      NOP   0;
//-InLocal---
      U     #tmpLocal;
      O     DB923.DBX 2509.1; // emergency regime without fan 2
      =     #A_3226_TSC01_AF.InLocal;
//
//-Monitoring---
      CLR   ;
      =     #A_3226_TSC01_AF.InMonLL;
      CLR   ;
      =     #A_3226_TSC01_AF.InMonL;
      CLR   ;
      =     #A_3226_TSC01_AF.InMonMid;
      CLR   ;
      =     #A_3226_TSC01_AF.InMonH;
      CLR   ;
      =     #A_3226_TSC01_AF.InMonHH;
//
//-Read inputs---
      L     #A_3226_TSC01_COM.InValuePC; // Umgerechnet in FU-FB
      T     #A_3226_TSC01_AF.InpValue;
      U     "PLC_SystemDB".GlobalFlags.Kilning_2;
      =     #A_3226_TSC01_AF.InHWStop;
//
//-Set Parameters---
// --> Erläuterung
      L     L#27648; // InpValue=Drehzahl direkt
      T     "G297M".A_3226_TSC01_AF.Par.ParUnitsByMaxDigit;
      L     L#10000; // OutValuePc=OutValueUnits
      T     "G297M".A_3226_TSC01_AF.Par.ParUnitsBy100Pc;
      L     L#4000; // 40.00% ist untere Grenze
      T     "G297M".A_3226_TSC01_AF.Par.ParLimitLL;
      L     L#4100; // 41.00%
      T     "G297M".A_3226_TSC01_AF.Par.ParLimitL;
      L     L#8000; // 80.00%
      T     "G297M".A_3226_TSC01_AF.Par.ParLimitH;
      L     L#10100; // 101.00%
      T     "G297M".A_3226_TSC01_AF.Par.ParLimitHH;
//
//-Call object control---
      CALL #A_3226_TSC01_AF ;
//
//-Write outputs---
NETWORK
TITLE ==A-3226-TSC01_AP : ACT. POWER FAN 2 FU

      NOP   0;
//-InLocal---
      U     #tmpLocal;
      O     DB923.DBX 2509.1; // emergency regime without fan 2
      =     #A_3226_TSC01_AP.InLocal;
//
//-Monitoring---
      CLR   ;
      =     #A_3226_TSC01_AP.InMonLL;
      CLR   ;
      =     #A_3226_TSC01_AP.InMonL;
      CLR   ;
      =     #A_3226_TSC01_AP.InMonMid;
      CLR   ;
      =     #A_3226_TSC01_AP.InMonH;
      CLR   ;
      =     #A_3226_TSC01_AP.InMonHH;
//
//-Read inputs---
      L     #A_3226_TSC01_COM.Output.SetpointValue03;
      T     #A_3226_TSC01_AP.InpValue;
      U     "PLC_SystemDB".GlobalFlags.Kilning_2;
      =     #A_3226_TSC01_AP.InHWStop;
//
//-Set Parameters---
// --> Erläuterung
      L     L#10650; // Leistung bei 27648Dez
      T     "G297M".A_3226_TSC01_AP.Par.ParUnitsByMaxDigit;
      L     L#10000; // OutValuePc=OutValueUnits
      T     "G297M".A_3226_TSC01_AP.Par.ParUnitsBy100Pc;
      L     L#0; // 0.0kW
      T     "G297M".A_3226_TSC01_AP.Par.ParLimitLL;
      L     L#100; // 10.0kW
      T     "G297M".A_3226_TSC01_AP.Par.ParLimitL;
      L     L#3150; // 315.0kW Motorleistung
      T     "G297M".A_3226_TSC01_AP.Par.ParLimitH;
      L     L#7000; // 631.1kW Leistung FU
      T     "G297M".A_3226_TSC01_AP.Par.ParLimitHH;
//
//-Call object control---
      CALL #A_3226_TSC01_AP ;
//
//-Write outputs---
NETWORK
TITLE ==A-3226-TSC01_AT : ACT. TORQUE FAN 2 FU

      NOP   0;
//-InLocal---
      U     #tmpLocal;
      O     DB923.DBX 2509.1; // emergency regime without fan 2
      =     #A_3226_TSC01_AT.InLocal;
//
//-Monitoring---
      CLR   ;
      =     #A_3226_TSC01_AT.InMonLL;
      CLR   ;
      =     #A_3226_TSC01_AT.InMonL;
      CLR   ;
      =     #A_3226_TSC01_AT.InMonMid;
      CLR   ;
      =     #A_3226_TSC01_AT.InMonH;
      CLR   ;
      =     #A_3226_TSC01_AT.InMonHH;
//
//-Read inputs---
      L     #A_3226_TSC01_COM.Output.SetpointValue04;
      L     0;
      U     #A_3226_TSC01_COM.Input.StateWord_1.BETRIEBSBEREIT;
      SPBN  M320;
      L     1500;
M320: T     #A_3226_TSC01_AT.InpValue;
      U     "PLC_SystemDB".GlobalFlags.Kilning_2;
      =     #A_3226_TSC01_AT.InHWStop;
//
//-Set Parameters---
// --> Erläuterung
      L     L#6835; // Drehmoment bei 27648Dez
      T     "G297M".A_3226_TSC01_AT.Par.ParUnitsByMaxDigit;
      L     L#10000; // OutValuePc=OutValueUnits
      T     "G297M".A_3226_TSC01_AT.Par.ParUnitsBy100Pc;
      L     L#0; // 0Nm
      T     "G297M".A_3226_TSC01_AT.Par.ParLimitLL;
      L     L#10; // 10Nm
      T     "G297M".A_3226_TSC01_AT.Par.ParLimitL;
      L     L#4050; // 4050Nm
      T     "G297M".A_3226_TSC01_AT.Par.ParLimitH;
      L     L#6835; // 6835Nm
      T     "G297M".A_3226_TSC01_AT.Par.ParLimitHH;
//
//-Call object control---
      CALL #A_3226_TSC01_AT ;
//
//-Write outputs---
NETWORK
TITLE ==A-3225-TSC01 : FAN 1 FU KOMMUNIKATION
NOP 0;
//-InLocal---
      U     #tmpLocal;
      =     #A_3225_TSC01.InLocal;
//
//-Monitoring---
      CLR;
      =      #A_3225_TSC01.InMonTrue;
      CLR;
      =      #A_3225_TSC01.InMonFalse;
//
//-PreAlarm---
      CLR;
      =      #A_3225_TSC01.InPreAlarmTrue;
      CLR;
      =      #A_3225_TSC01.InPreAlarmFalse;
//
//-Additional commands---
//      CLR
//      S     #A_3225_TSC01.CmdRunTimeOutTime
//
//-Read inputs---
      U     M 050.0;
      =     #A_3225_TSC01.InpTrue;
//
//-Set Parameters---
//
//-Call object control---
      CALL  #A_3225_TSC01;
//
//-Write outputs---
NETWORK
TITLE =Test Fault
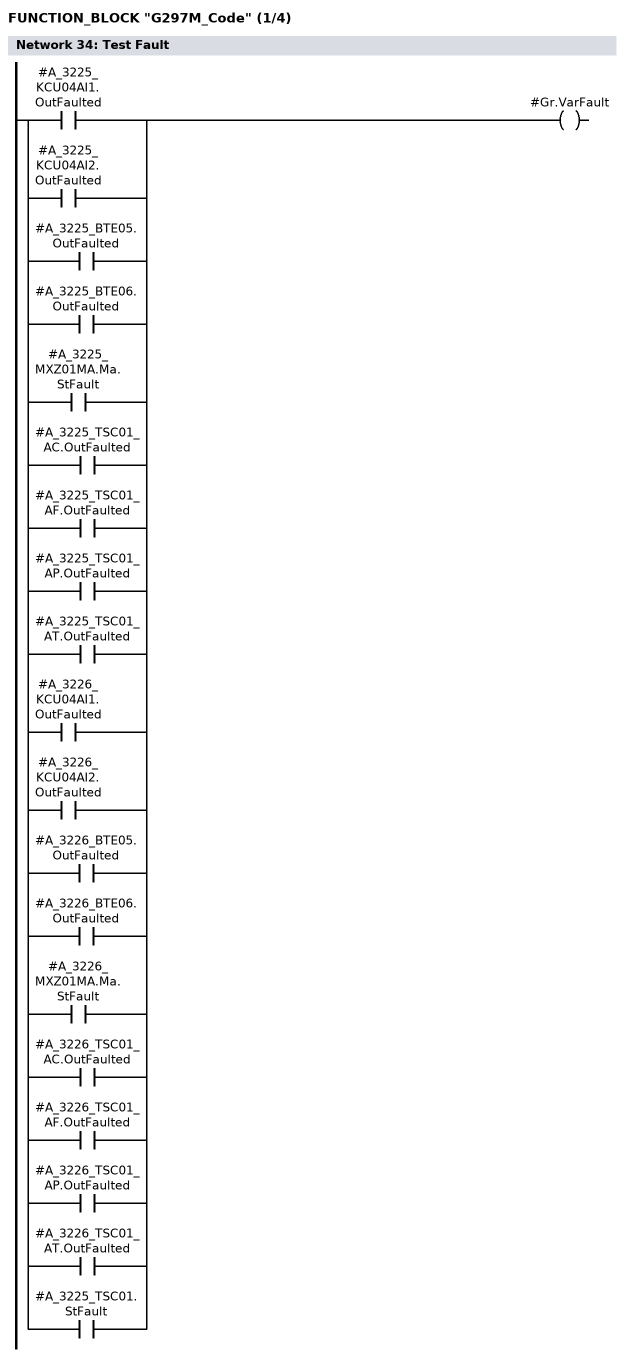

      U     #A_3225_KCU04AI1.OutFaulted;
      O     #A_3225_KCU04AI2.OutFaulted;
      O     #A_3225_BTE05.OutFaulted;
      O     #A_3225_BTE06.OutFaulted;
      O     #A_3225_MXZ01MA.Ma.StFault;
      O     #A_3225_TSC01_AC.OutFaulted;
      O     #A_3225_TSC01_AF.OutFaulted;
      O     #A_3225_TSC01_AP.OutFaulted;
      O     #A_3225_TSC01_AT.OutFaulted;
      O     #A_3226_KCU04AI1.OutFaulted;
      O     #A_3226_KCU04AI2.OutFaulted;
      O     #A_3226_BTE05.OutFaulted;
      O     #A_3226_BTE06.OutFaulted;
      O     #A_3226_MXZ01MA.Ma.StFault;
      O     #A_3226_TSC01_AC.OutFaulted;
      O     #A_3226_TSC01_AF.OutFaulted;
      O     #A_3226_TSC01_AP.OutFaulted;
      O     #A_3226_TSC01_AT.OutFaulted;
      O     #A_3225_TSC01.StFault;
      =     #Gr.VarFault;
NETWORK
TITLE =Test Warning
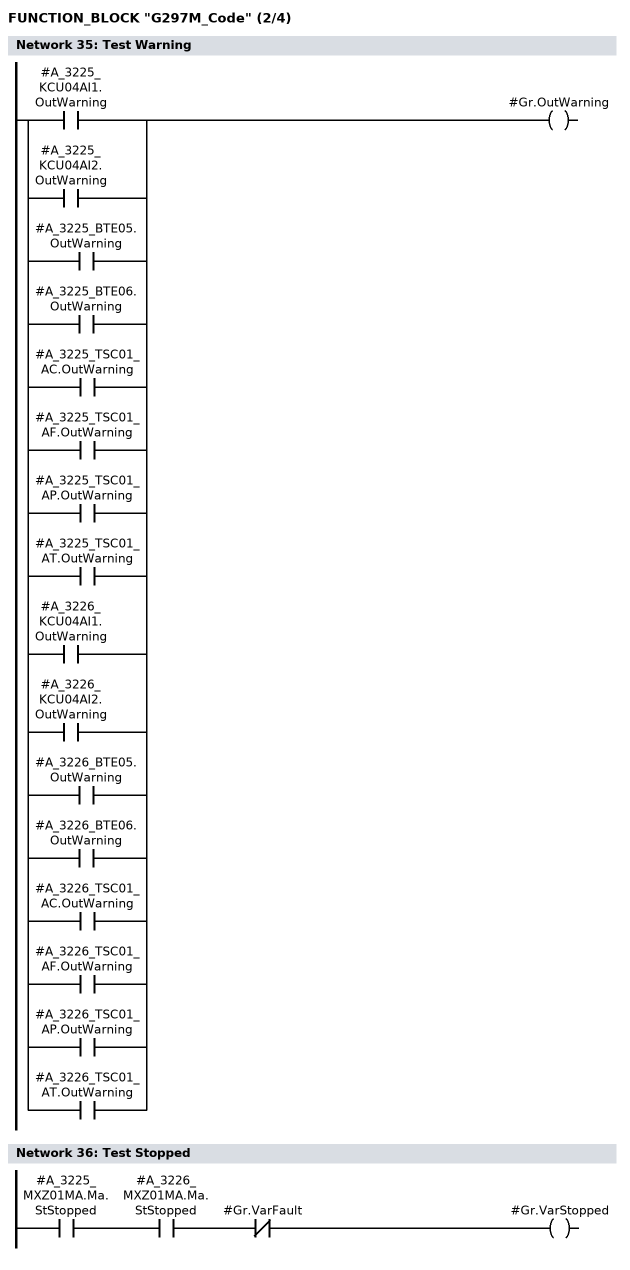

      U     #A_3225_KCU04AI1.OutWarning;
      O     #A_3225_KCU04AI2.OutWarning;
      O     #A_3225_BTE05.OutWarning;
      O     #A_3225_BTE06.OutWarning;
      O     #A_3225_TSC01_AC.OutWarning;
      O     #A_3225_TSC01_AF.OutWarning;
      O     #A_3225_TSC01_AP.OutWarning;
      O     #A_3225_TSC01_AT.OutWarning;
      O     #A_3226_KCU04AI1.OutWarning;
      O     #A_3226_KCU04AI2.OutWarning;
      O     #A_3226_BTE05.OutWarning;
      O     #A_3226_BTE06.OutWarning;
      O     #A_3226_TSC01_AC.OutWarning;
      O     #A_3226_TSC01_AF.OutWarning;
      O     #A_3226_TSC01_AP.OutWarning;
      O     #A_3226_TSC01_AT.OutWarning;
      =     #Gr.OutWarning;
NETWORK
TITLE =Test Stopped

      U     #A_3225_MXZ01MA.Ma.StStopped;
      U     #A_3226_MXZ01MA.Ma.StStopped;
      UN    #Gr.VarFault;
      =     #Gr.VarStopped;
NETWORK
TITLE =Test Started
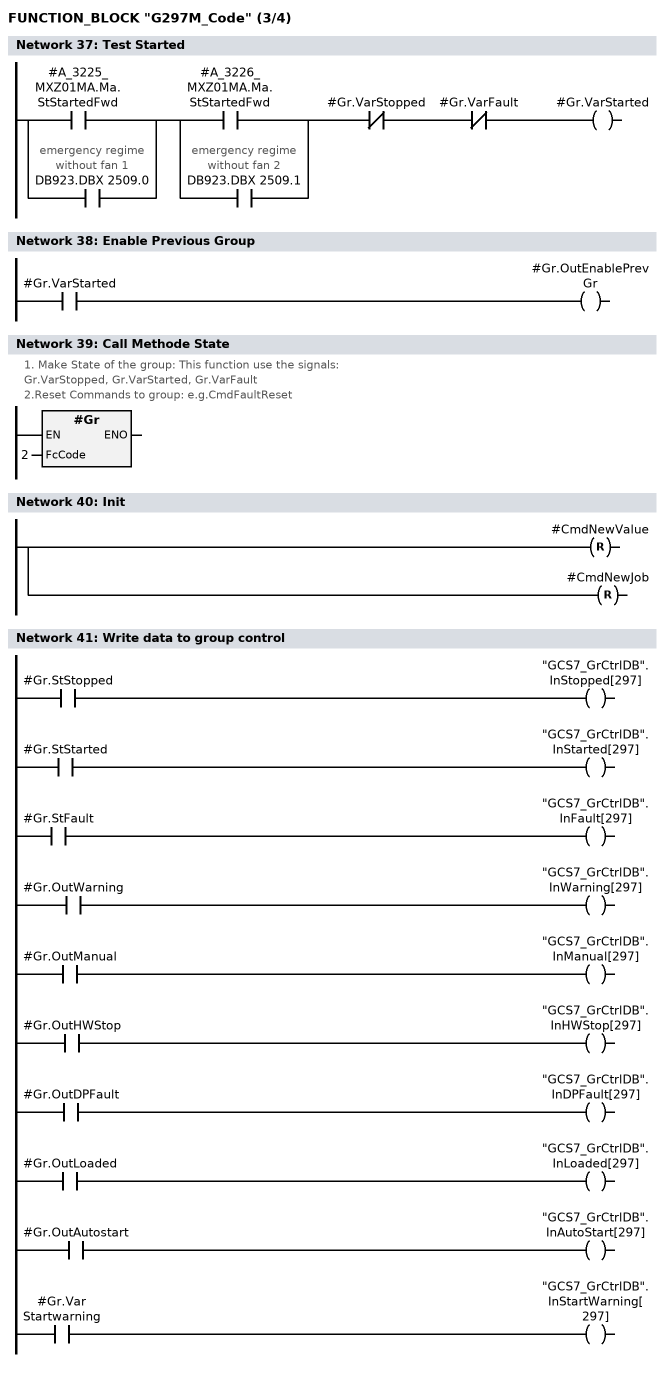

      U(    ;
      U     #A_3225_MXZ01MA.Ma.StStartedFwd;
      O     DB923.DBX 2509.0; // emergency regime without fan 1
      )     ;
      U(    ;
      U     #A_3226_MXZ01MA.Ma.StStartedFwd;
      O     DB923.DBX 2509.1; // emergency regime without fan 2
      )     ;
      UN    #Gr.VarStopped;
      UN    #Gr.VarFault;
      =     #Gr.VarStarted;
NETWORK
TITLE =Enable Previous Group

      U     #Gr.VarStarted;
      =     #Gr.OutEnablePrevGr;
NETWORK
TITLE =Call Methode State
//1. Make State of the group: This function use the signals:
//        Gr.VarStopped, Gr.VarStarted, Gr.VarFault
//2.Reset Commands to group: e.g.CmdFaultReset
      CALL #Gr (
           FcCode                   := 2);
NETWORK
TITLE =Init

      SET   ;
      R     #CmdNewValue;
      R     #CmdNewJob;
NETWORK
TITLE =Write data to group control

      U     #Gr.StStopped;
      =     "GCS7_GrCtrlDB".InStopped[297];
      U     #Gr.StStarted;
      =     "GCS7_GrCtrlDB".InStarted[297];
      U     #Gr.StFault;
      =     "GCS7_GrCtrlDB".InFault[297];
      U     #Gr.OutWarning;
      =     "GCS7_GrCtrlDB".InWarning[297];
      U     #Gr.OutManual;
      =     "GCS7_GrCtrlDB".InManual[297];
      U     #Gr.OutHWStop;
      =     "GCS7_GrCtrlDB".InHWStop[297];
      U     #Gr.OutDPFault;
      =     "GCS7_GrCtrlDB".InDPFault[297];
      U     #Gr.OutLoaded;
      =     "GCS7_GrCtrlDB".InLoaded[297];
      U     #Gr.OutAutostart;
      =     "GCS7_GrCtrlDB".InAutoStart[297];
      U     #Gr.VarStartwarning;
      =     "GCS7_GrCtrlDB".InStartWarning[297];
NETWORK
TITLE =End of block
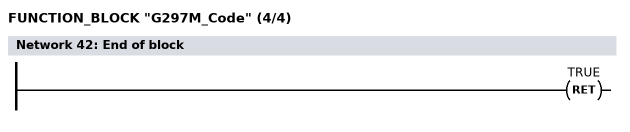

      BE    ;

END_FUNCTION_BLOCK


DATA_BLOCK "G297M"
TITLE =DBG297M  FAN KILN 2
//COPYRIGHT:    (C) 2009  BUHLER AG, CH-9240 UZWIL, SWITZERLAND
//
//PRODUCT:      WinCoS_BIW01_09
//
//TITLE:        FAN KILN 2
//                Machine group DB
//                Maschinengruppen-DB
//
//-------------------------------------------------------------------------
//
//IDENT:        AUTHOR:             DEPT:             DATE:
//
//P01_DB397.1.0 K.Renz              CSB41             09.Okt.2009
//              1st Release
//
//-------------------------------------------------------------------------
//
//PURPOSE:
//
//MANUAL :
//
//RESTRICTIONS:
//
//-------------------------------------------------------------------------
AUTHOR : KR
FAMILY : USW
NAME : DBG297M
VERSION : 0.0

"G297M_Code"
BEGIN
   Gr.FcCode := 0;
   Gr.Spare2 := 0;
   Gr.Spare4 := 0;
   Gr.Spare6 := 0;
   Gr.OutEmptyingTime := 0;
   Gr.ChangeBit.spare := B#16#0;
   Gr.ChangeBit.CBit1 := FALSE;
   Gr.ChangeBit.CBit2 := FALSE;
   Gr.ChangeBit.CBit3 := FALSE;
   Gr.ChangeBit.CBit4 := FALSE;
   Gr.StCode := 0;
   Gr.InEnableGr := FALSE;
   Gr.CmdContinue := FALSE;
   Gr.CmdRestartIdling := FALSE;
   Gr.InReleaseEmptyingTime := FALSE;
   Gr.InFeeding := FALSE;
   Gr.InOutAutostartMan := FALSE;
   Gr.InPreStart := FALSE;
   Gr.CmdManualOff := FALSE;
   Gr.CmdOff := FALSE;
   Gr.CmdOn := FALSE;
   Gr.CmdNext := FALSE;
   Gr.CmdFaultReset := FALSE;
   Gr.InOccupied := FALSE;
   Gr.InManual := FALSE;
   Gr.InLoadedSec := FALSE;
   Gr.InSeqStop := FALSE;
   Gr.ModePassive := FALSE;
   Gr.ModeActive := FALSE;
   Gr.ModeIdling := FALSE;
   Gr.spare163 := FALSE;
   Gr.spare164 := FALSE;
   Gr.spare165 := FALSE;
   Gr.spare166 := FALSE;
   Gr.spare167 := FALSE;
   Gr.StStopped := FALSE;
   Gr.StStarting := FALSE;
   Gr.StStarted := FALSE;
   Gr.StStopping := FALSE;
   Gr.StFault := FALSE;
   Gr.OutLoaded := FALSE;
   Gr.OutWarning := FALSE;
   Gr.OutFeeding := FALSE;
   Gr.OutEnableEl := FALSE;
   Gr.OutEnable1 := FALSE;
   Gr.OutHWStop := FALSE;
   Gr.OutDPFault := FALSE;
   Gr.OutAutostart := FALSE;
   Gr.OutManual := FALSE;
   Gr.OutHornOn := FALSE;
   Gr.OutEnablePrevGr := FALSE;
   Gr.VarStopped := FALSE;
   Gr.VarStarted := FALSE;
   Gr.VarFault := FALSE;
   Gr.VarStartwarning := FALSE;
   Gr.VarFlag1s := FALSE;
   Gr.OutEmptyingTimeDone := FALSE;
   Gr.OutNewWay := FALSE;
   Gr.OutSeqStop := FALSE;
   Gr.OutIdlingTime := 0;
   Gr.InCodePreselect := 0;
   Gr.InLine := 0;
   Gr.InCode := 0;
   Gr.OutCode := 0;
   Gr.Par.ParObjectNo := 29700;
   Gr.Par.ParMgr := TRUE;
   Gr.Par.ParWgr := FALSE;
   Gr.Par.ParGgr := FALSE;
   Gr.Par.ParHornCode := 11;
   Gr.Par.ParIdling := 2;
   Gr.Par.ParEmptyingTime := 0;
   Gr.Par.Para1_0 := FALSE;
   Gr.Par.Para1_1 := FALSE;
   Gr.Par.Para1_2 := FALSE;
   Gr.Par.Para1_3 := FALSE;
   Gr.Par.Para1_4 := FALSE;
   Gr.Par.Para1_5 := FALSE;
   Gr.Par.Para1_6 := FALSE;
   Gr.Par.Para1_7 := FALSE;
   Gr.Par.Para1_8 := FALSE;
   Gr.Par.Para1_9 := FALSE;
   Gr.Par.Para1_10 := FALSE;
   Gr.Par.Para1_11 := FALSE;
   Gr.Par.Para1_12 := FALSE;
   Gr.Par.Para1_13 := FALSE;
   Gr.Par.Para1_14 := FALSE;
   Gr.Par.Para1_15 := FALSE;
   Gr.Par.Para2 := 0;
   Gr.Par.Para3 := 0;
   Gr.Par.Para4 := 0;
   Gr.Par.Para5 := 0;
   InOutValue1 := L#0;
   InOutValue2 := L#0;
   OutWayConflict := FALSE;
   OutSelectionOk := FALSE;
   CmdNewValue := FALSE;
   CmdNewJob := FALSE;
   OutCodeOK := FALSE;
   InEndOfJob := FALSE;
   staWayOk := FALSE;
   EdgeStartRelease := FALSE;
   USW8 := FALSE;
   USW9 := FALSE;
   USW10 := FALSE;
   USW11 := FALSE;
   USW12 := FALSE;
   USW13 := FALSE;
   USW14 := FALSE;
   USW15 := FALSE;
   A_3225_KCU04AI1.StCode := 0;
   A_3225_KCU04AI1.InMonLL := FALSE;
   A_3225_KCU04AI1.InMonL := FALSE;
   A_3225_KCU04AI1.InMonMid := FALSE;
   A_3225_KCU04AI1.InMonH := FALSE;
   A_3225_KCU04AI1.InMonHH := FALSE;
   A_3225_KCU04AI1.spare0205 := FALSE;
   A_3225_KCU04AI1.InpFaultAI := FALSE;
   A_3225_KCU04AI1.InpFaultDev := FALSE;
   A_3225_KCU04AI1.InHWStop := FALSE;
   A_3225_KCU04AI1.InDPFault := FALSE;
   A_3225_KCU04AI1.InDisable := FALSE;
   A_3225_KCU04AI1.CmdFaultReset := FALSE;
   A_3225_KCU04AI1.InLocal := FALSE;
   A_3225_KCU04AI1.spare0305 := FALSE;
   A_3225_KCU04AI1.InReport := FALSE;
   A_3225_KCU04AI1.spare0307 := FALSE;
   A_3225_KCU04AI1.OutLL := FALSE;
   A_3225_KCU04AI1.OutL := FALSE;
   A_3225_KCU04AI1.OutH := FALSE;
   A_3225_KCU04AI1.OutHH := FALSE;
   A_3225_KCU04AI1.OutOverflow := FALSE;
   A_3225_KCU04AI1.spare0405 := FALSE;
   A_3225_KCU04AI1.OutFaultAI := FALSE;
   A_3225_KCU04AI1.spare0407 := FALSE;
   A_3225_KCU04AI1.StLL := FALSE;
   A_3225_KCU04AI1.StL := FALSE;
   A_3225_KCU04AI1.StMid := FALSE;
   A_3225_KCU04AI1.StH := FALSE;
   A_3225_KCU04AI1.StHH := FALSE;
   A_3225_KCU04AI1.StFaultAI := FALSE;
   A_3225_KCU04AI1.OutWarning := FALSE;
   A_3225_KCU04AI1.OutFaulted := FALSE;
   A_3225_KCU04AI1.InpValue := 0;
   A_3225_KCU04AI1.OutValuePc := 0;
   A_3225_KCU04AI1.OutValueUnits := L#0;
   A_3225_KCU04AI1.Msg.WarningDoneLL := FALSE;
   A_3225_KCU04AI1.Msg.WarningDoneL := FALSE;
   A_3225_KCU04AI1.Msg.WarningDoneMid := FALSE;
   A_3225_KCU04AI1.Msg.WarningDoneH := FALSE;
   A_3225_KCU04AI1.Msg.WarningDoneHH := FALSE;
   A_3225_KCU04AI1.Msg.FaultDoneLL := FALSE;
   A_3225_KCU04AI1.Msg.FaultDoneL := FALSE;
   A_3225_KCU04AI1.Msg.FaultDoneMid := FALSE;
   A_3225_KCU04AI1.Msg.FaultDoneH := FALSE;
   A_3225_KCU04AI1.Msg.FaultDoneHH := FALSE;
   A_3225_KCU04AI1.Msg.FaultDoneDev := FALSE;
   A_3225_KCU04AI1.Msg.FaultDoneAI := FALSE;
   A_3225_KCU04AI1.OutAlarmNrLog := 0;
   A_3225_KCU04AI1.Par.ParObjectNo := 29701;
   A_3225_KCU04AI1.Par.ParMsgType := 7252;
   A_3225_KCU04AI1.Par.ParHornCode := 11;
   A_3225_KCU04AI1.Par.ParLogOff := FALSE;
   A_3225_KCU04AI1.Par.ParSpare0401 := FALSE;
   A_3225_KCU04AI1.Par.ParValueByUser := FALSE;
   A_3225_KCU04AI1.Par.ParLimitsPc := TRUE;
   A_3225_KCU04AI1.Par.ParWago := FALSE;
   A_3225_KCU04AI1.Par.ParNoHornByWarning := FALSE;
   A_3225_KCU04AI1.Par.ParWarningLL := FALSE;
   A_3225_KCU04AI1.Par.ParWarningL := FALSE;
   A_3225_KCU04AI1.Par.ParWarningMid := FALSE;
   A_3225_KCU04AI1.Par.ParWarningH := TRUE;
   A_3225_KCU04AI1.Par.ParWarningHH := FALSE;
   A_3225_KCU04AI1.Par.ParPreAlarmLL := FALSE;
   A_3225_KCU04AI1.Par.ParPreAlarmL := FALSE;
   A_3225_KCU04AI1.Par.ParPreAlarmMid := FALSE;
   A_3225_KCU04AI1.Par.ParPreAlarmH := FALSE;
   A_3225_KCU04AI1.Par.ParPreAlarmHH := FALSE;
   A_3225_KCU04AI1.Par.ParUnitsByZeroDigit := L#0;
   A_3225_KCU04AI1.Par.ParUnitsByMaxDigit := L#2000;
   A_3225_KCU04AI1.Par.ParUnitsBy100Pc := L#10000;
   A_3225_KCU04AI1.Par.ParLimitLL := L#-1;
   A_3225_KCU04AI1.Par.ParLimitL := L#0;
   A_3225_KCU04AI1.Par.ParLimitH := L#3150;
   A_3225_KCU04AI1.Par.ParLimitHH := L#3550;
   A_3225_KCU04AI1.Par.ParMonTimeLL := 0;
   A_3225_KCU04AI1.Par.ParMonTimeL := 0;
   A_3225_KCU04AI1.Par.ParMonTimeMid := 0;
   A_3225_KCU04AI1.Par.ParMonTimeH := 600;
   A_3225_KCU04AI1.Par.ParMonTimeHH := 0;
   A_3225_KCU04AI1.Par.ParDelayTimeDown := 10;
   A_3225_KCU04AI1.Par.ParDelayTimeUp := 10;
   A_3225_KCU04AI1.Par.ParDelayTime := 30;
   A_3225_KCU04AI1.Par.OutMonTimeLL := 0;
   A_3225_KCU04AI1.Par.OutMonTimeL := 0;
   A_3225_KCU04AI1.Par.OutMonTimeMid := 0;
   A_3225_KCU04AI1.Par.OutMonTimeH := 0;
   A_3225_KCU04AI1.Par.OutMonTimeHH := 0;
   A_3225_KCU04AI1.Par.OutDelayTimeDown := 0;
   A_3225_KCU04AI1.Par.OutDelayTimeUp := 0;
   A_3225_KCU04AI1.Par.OutDelayTime := 0;
   A_3225_KCU04AI1.Par.Spare66 := 0;
   A_3225_KCU04AI2.StCode := 0;
   A_3225_KCU04AI2.InMonLL := FALSE;
   A_3225_KCU04AI2.InMonL := FALSE;
   A_3225_KCU04AI2.InMonMid := FALSE;
   A_3225_KCU04AI2.InMonH := FALSE;
   A_3225_KCU04AI2.InMonHH := FALSE;
   A_3225_KCU04AI2.spare0205 := FALSE;
   A_3225_KCU04AI2.InpFaultAI := FALSE;
   A_3225_KCU04AI2.InpFaultDev := FALSE;
   A_3225_KCU04AI2.InHWStop := FALSE;
   A_3225_KCU04AI2.InDPFault := FALSE;
   A_3225_KCU04AI2.InDisable := FALSE;
   A_3225_KCU04AI2.CmdFaultReset := FALSE;
   A_3225_KCU04AI2.InLocal := FALSE;
   A_3225_KCU04AI2.spare0305 := FALSE;
   A_3225_KCU04AI2.InReport := FALSE;
   A_3225_KCU04AI2.spare0307 := FALSE;
   A_3225_KCU04AI2.OutLL := FALSE;
   A_3225_KCU04AI2.OutL := FALSE;
   A_3225_KCU04AI2.OutH := FALSE;
   A_3225_KCU04AI2.OutHH := FALSE;
   A_3225_KCU04AI2.OutOverflow := FALSE;
   A_3225_KCU04AI2.spare0405 := FALSE;
   A_3225_KCU04AI2.OutFaultAI := FALSE;
   A_3225_KCU04AI2.spare0407 := FALSE;
   A_3225_KCU04AI2.StLL := FALSE;
   A_3225_KCU04AI2.StL := FALSE;
   A_3225_KCU04AI2.StMid := FALSE;
   A_3225_KCU04AI2.StH := FALSE;
   A_3225_KCU04AI2.StHH := FALSE;
   A_3225_KCU04AI2.StFaultAI := FALSE;
   A_3225_KCU04AI2.OutWarning := FALSE;
   A_3225_KCU04AI2.OutFaulted := FALSE;
   A_3225_KCU04AI2.InpValue := 0;
   A_3225_KCU04AI2.OutValuePc := 0;
   A_3225_KCU04AI2.OutValueUnits := L#0;
   A_3225_KCU04AI2.Msg.WarningDoneLL := FALSE;
   A_3225_KCU04AI2.Msg.WarningDoneL := FALSE;
   A_3225_KCU04AI2.Msg.WarningDoneMid := FALSE;
   A_3225_KCU04AI2.Msg.WarningDoneH := FALSE;
   A_3225_KCU04AI2.Msg.WarningDoneHH := FALSE;
   A_3225_KCU04AI2.Msg.FaultDoneLL := FALSE;
   A_3225_KCU04AI2.Msg.FaultDoneL := FALSE;
   A_3225_KCU04AI2.Msg.FaultDoneMid := FALSE;
   A_3225_KCU04AI2.Msg.FaultDoneH := FALSE;
   A_3225_KCU04AI2.Msg.FaultDoneHH := FALSE;
   A_3225_KCU04AI2.Msg.FaultDoneDev := FALSE;
   A_3225_KCU04AI2.Msg.FaultDoneAI := FALSE;
   A_3225_KCU04AI2.OutAlarmNrLog := 0;
   A_3225_KCU04AI2.Par.ParObjectNo := 29702;
   A_3225_KCU04AI2.Par.ParMsgType := 7252;
   A_3225_KCU04AI2.Par.ParHornCode := 11;
   A_3225_KCU04AI2.Par.ParLogOff := FALSE;
   A_3225_KCU04AI2.Par.ParSpare0401 := FALSE;
   A_3225_KCU04AI2.Par.ParValueByUser := FALSE;
   A_3225_KCU04AI2.Par.ParLimitsPc := TRUE;
   A_3225_KCU04AI2.Par.ParWago := FALSE;
   A_3225_KCU04AI2.Par.ParNoHornByWarning := FALSE;
   A_3225_KCU04AI2.Par.ParWarningLL := FALSE;
   A_3225_KCU04AI2.Par.ParWarningL := FALSE;
   A_3225_KCU04AI2.Par.ParWarningMid := FALSE;
   A_3225_KCU04AI2.Par.ParWarningH := TRUE;
   A_3225_KCU04AI2.Par.ParWarningHH := FALSE;
   A_3225_KCU04AI2.Par.ParPreAlarmLL := FALSE;
   A_3225_KCU04AI2.Par.ParPreAlarmL := FALSE;
   A_3225_KCU04AI2.Par.ParPreAlarmMid := FALSE;
   A_3225_KCU04AI2.Par.ParPreAlarmH := FALSE;
   A_3225_KCU04AI2.Par.ParPreAlarmHH := FALSE;
   A_3225_KCU04AI2.Par.ParUnitsByZeroDigit := L#0;
   A_3225_KCU04AI2.Par.ParUnitsByMaxDigit := L#2000;
   A_3225_KCU04AI2.Par.ParUnitsBy100Pc := L#10000;
   A_3225_KCU04AI2.Par.ParLimitLL := L#-1;
   A_3225_KCU04AI2.Par.ParLimitL := L#0;
   A_3225_KCU04AI2.Par.ParLimitH := L#3150;
   A_3225_KCU04AI2.Par.ParLimitHH := L#3550;
   A_3225_KCU04AI2.Par.ParMonTimeLL := 0;
   A_3225_KCU04AI2.Par.ParMonTimeL := 0;
   A_3225_KCU04AI2.Par.ParMonTimeMid := 0;
   A_3225_KCU04AI2.Par.ParMonTimeH := 600;
   A_3225_KCU04AI2.Par.ParMonTimeHH := 0;
   A_3225_KCU04AI2.Par.ParDelayTimeDown := 10;
   A_3225_KCU04AI2.Par.ParDelayTimeUp := 10;
   A_3225_KCU04AI2.Par.ParDelayTime := 30;
   A_3225_KCU04AI2.Par.OutMonTimeLL := 0;
   A_3225_KCU04AI2.Par.OutMonTimeL := 0;
   A_3225_KCU04AI2.Par.OutMonTimeMid := 0;
   A_3225_KCU04AI2.Par.OutMonTimeH := 0;
   A_3225_KCU04AI2.Par.OutMonTimeHH := 0;
   A_3225_KCU04AI2.Par.OutDelayTimeDown := 0;
   A_3225_KCU04AI2.Par.OutDelayTimeUp := 0;
   A_3225_KCU04AI2.Par.OutDelayTime := 0;
   A_3225_KCU04AI2.Par.Spare66 := 0;
   A_3225_BTE05.StCode := 0;
   A_3225_BTE05.InMonLL := FALSE;
   A_3225_BTE05.InMonL := FALSE;
   A_3225_BTE05.InMonMid := FALSE;
   A_3225_BTE05.InMonH := FALSE;
   A_3225_BTE05.InMonHH := FALSE;
   A_3225_BTE05.spare0205 := FALSE;
   A_3225_BTE05.InpFaultAI := FALSE;
   A_3225_BTE05.InpFaultDev := FALSE;
   A_3225_BTE05.InHWStop := FALSE;
   A_3225_BTE05.InDPFault := FALSE;
   A_3225_BTE05.InDisable := FALSE;
   A_3225_BTE05.CmdFaultReset := FALSE;
   A_3225_BTE05.InLocal := FALSE;
   A_3225_BTE05.spare0305 := FALSE;
   A_3225_BTE05.InReport := FALSE;
   A_3225_BTE05.spare0307 := FALSE;
   A_3225_BTE05.OutLL := FALSE;
   A_3225_BTE05.OutL := FALSE;
   A_3225_BTE05.OutH := FALSE;
   A_3225_BTE05.OutHH := FALSE;
   A_3225_BTE05.OutOverflow := FALSE;
   A_3225_BTE05.spare0405 := FALSE;
   A_3225_BTE05.OutFaultAI := FALSE;
   A_3225_BTE05.spare0407 := FALSE;
   A_3225_BTE05.StLL := FALSE;
   A_3225_BTE05.StL := FALSE;
   A_3225_BTE05.StMid := FALSE;
   A_3225_BTE05.StH := FALSE;
   A_3225_BTE05.StHH := FALSE;
   A_3225_BTE05.StFaultAI := FALSE;
   A_3225_BTE05.OutWarning := FALSE;
   A_3225_BTE05.OutFaulted := FALSE;
   A_3225_BTE05.InpValue := 0;
   A_3225_BTE05.OutValuePc := 0;
   A_3225_BTE05.OutValueUnits := L#0;
   A_3225_BTE05.Msg.WarningDoneLL := FALSE;
   A_3225_BTE05.Msg.WarningDoneL := FALSE;
   A_3225_BTE05.Msg.WarningDoneMid := FALSE;
   A_3225_BTE05.Msg.WarningDoneH := FALSE;
   A_3225_BTE05.Msg.WarningDoneHH := FALSE;
   A_3225_BTE05.Msg.FaultDoneLL := FALSE;
   A_3225_BTE05.Msg.FaultDoneL := FALSE;
   A_3225_BTE05.Msg.FaultDoneMid := FALSE;
   A_3225_BTE05.Msg.FaultDoneH := FALSE;
   A_3225_BTE05.Msg.FaultDoneHH := FALSE;
   A_3225_BTE05.Msg.FaultDoneDev := FALSE;
   A_3225_BTE05.Msg.FaultDoneAI := FALSE;
   A_3225_BTE05.OutAlarmNrLog := 0;
   A_3225_BTE05.Par.ParObjectNo := 29703;
   A_3225_BTE05.Par.ParMsgType := 7252;
   A_3225_BTE05.Par.ParHornCode := 11;
   A_3225_BTE05.Par.ParLogOff := FALSE;
   A_3225_BTE05.Par.ParSpare0401 := FALSE;
   A_3225_BTE05.Par.ParValueByUser := FALSE;
   A_3225_BTE05.Par.ParLimitsPc := TRUE;
   A_3225_BTE05.Par.ParWago := FALSE;
   A_3225_BTE05.Par.ParNoHornByWarning := FALSE;
   A_3225_BTE05.Par.ParWarningLL := FALSE;
   A_3225_BTE05.Par.ParWarningL := FALSE;
   A_3225_BTE05.Par.ParWarningMid := FALSE;
   A_3225_BTE05.Par.ParWarningH := TRUE;
   A_3225_BTE05.Par.ParWarningHH := FALSE;
   A_3225_BTE05.Par.ParPreAlarmLL := FALSE;
   A_3225_BTE05.Par.ParPreAlarmL := FALSE;
   A_3225_BTE05.Par.ParPreAlarmMid := FALSE;
   A_3225_BTE05.Par.ParPreAlarmH := FALSE;
   A_3225_BTE05.Par.ParPreAlarmHH := FALSE;
   A_3225_BTE05.Par.ParUnitsByZeroDigit := L#0;
   A_3225_BTE05.Par.ParUnitsByMaxDigit := L#27384;
   A_3225_BTE05.Par.ParUnitsBy100Pc := L#10000;
   A_3225_BTE05.Par.ParLimitLL := L#0;
   A_3225_BTE05.Par.ParLimitL := L#2000;
   A_3225_BTE05.Par.ParLimitH := L#8000;
   A_3225_BTE05.Par.ParLimitHH := L#10000;
   A_3225_BTE05.Par.ParMonTimeLL := 0;
   A_3225_BTE05.Par.ParMonTimeL := 0;
   A_3225_BTE05.Par.ParMonTimeMid := 0;
   A_3225_BTE05.Par.ParMonTimeH := 600;
   A_3225_BTE05.Par.ParMonTimeHH := 0;
   A_3225_BTE05.Par.ParDelayTimeDown := 10;
   A_3225_BTE05.Par.ParDelayTimeUp := 10;
   A_3225_BTE05.Par.ParDelayTime := 30;
   A_3225_BTE05.Par.OutMonTimeLL := 0;
   A_3225_BTE05.Par.OutMonTimeL := 0;
   A_3225_BTE05.Par.OutMonTimeMid := 0;
   A_3225_BTE05.Par.OutMonTimeH := 0;
   A_3225_BTE05.Par.OutMonTimeHH := 0;
   A_3225_BTE05.Par.OutDelayTimeDown := 0;
   A_3225_BTE05.Par.OutDelayTimeUp := 0;
   A_3225_BTE05.Par.OutDelayTime := 0;
   A_3225_BTE05.Par.Spare66 := 0;
   A_3225_BTE06.StCode := 0;
   A_3225_BTE06.InMonLL := FALSE;
   A_3225_BTE06.InMonL := FALSE;
   A_3225_BTE06.InMonMid := FALSE;
   A_3225_BTE06.InMonH := FALSE;
   A_3225_BTE06.InMonHH := FALSE;
   A_3225_BTE06.spare0205 := FALSE;
   A_3225_BTE06.InpFaultAI := FALSE;
   A_3225_BTE06.InpFaultDev := FALSE;
   A_3225_BTE06.InHWStop := FALSE;
   A_3225_BTE06.InDPFault := FALSE;
   A_3225_BTE06.InDisable := FALSE;
   A_3225_BTE06.CmdFaultReset := FALSE;
   A_3225_BTE06.InLocal := FALSE;
   A_3225_BTE06.spare0305 := FALSE;
   A_3225_BTE06.InReport := FALSE;
   A_3225_BTE06.spare0307 := FALSE;
   A_3225_BTE06.OutLL := FALSE;
   A_3225_BTE06.OutL := FALSE;
   A_3225_BTE06.OutH := FALSE;
   A_3225_BTE06.OutHH := FALSE;
   A_3225_BTE06.OutOverflow := FALSE;
   A_3225_BTE06.spare0405 := FALSE;
   A_3225_BTE06.OutFaultAI := FALSE;
   A_3225_BTE06.spare0407 := FALSE;
   A_3225_BTE06.StLL := FALSE;
   A_3225_BTE06.StL := FALSE;
   A_3225_BTE06.StMid := FALSE;
   A_3225_BTE06.StH := FALSE;
   A_3225_BTE06.StHH := FALSE;
   A_3225_BTE06.StFaultAI := FALSE;
   A_3225_BTE06.OutWarning := FALSE;
   A_3225_BTE06.OutFaulted := FALSE;
   A_3225_BTE06.InpValue := 0;
   A_3225_BTE06.OutValuePc := 0;
   A_3225_BTE06.OutValueUnits := L#0;
   A_3225_BTE06.Msg.WarningDoneLL := FALSE;
   A_3225_BTE06.Msg.WarningDoneL := FALSE;
   A_3225_BTE06.Msg.WarningDoneMid := FALSE;
   A_3225_BTE06.Msg.WarningDoneH := FALSE;
   A_3225_BTE06.Msg.WarningDoneHH := FALSE;
   A_3225_BTE06.Msg.FaultDoneLL := FALSE;
   A_3225_BTE06.Msg.FaultDoneL := FALSE;
   A_3225_BTE06.Msg.FaultDoneMid := FALSE;
   A_3225_BTE06.Msg.FaultDoneH := FALSE;
   A_3225_BTE06.Msg.FaultDoneHH := FALSE;
   A_3225_BTE06.Msg.FaultDoneDev := FALSE;
   A_3225_BTE06.Msg.FaultDoneAI := FALSE;
   A_3225_BTE06.OutAlarmNrLog := 0;
   A_3225_BTE06.Par.ParObjectNo := 29704;
   A_3225_BTE06.Par.ParMsgType := 7252;
   A_3225_BTE06.Par.ParHornCode := 11;
   A_3225_BTE06.Par.ParLogOff := FALSE;
   A_3225_BTE06.Par.ParSpare0401 := FALSE;
   A_3225_BTE06.Par.ParValueByUser := FALSE;
   A_3225_BTE06.Par.ParLimitsPc := TRUE;
   A_3225_BTE06.Par.ParWago := FALSE;
   A_3225_BTE06.Par.ParNoHornByWarning := FALSE;
   A_3225_BTE06.Par.ParWarningLL := FALSE;
   A_3225_BTE06.Par.ParWarningL := FALSE;
   A_3225_BTE06.Par.ParWarningMid := FALSE;
   A_3225_BTE06.Par.ParWarningH := TRUE;
   A_3225_BTE06.Par.ParWarningHH := FALSE;
   A_3225_BTE06.Par.ParPreAlarmLL := FALSE;
   A_3225_BTE06.Par.ParPreAlarmL := FALSE;
   A_3225_BTE06.Par.ParPreAlarmMid := FALSE;
   A_3225_BTE06.Par.ParPreAlarmH := FALSE;
   A_3225_BTE06.Par.ParPreAlarmHH := FALSE;
   A_3225_BTE06.Par.ParUnitsByZeroDigit := L#0;
   A_3225_BTE06.Par.ParUnitsByMaxDigit := L#27384;
   A_3225_BTE06.Par.ParUnitsBy100Pc := L#10000;
   A_3225_BTE06.Par.ParLimitLL := L#0;
   A_3225_BTE06.Par.ParLimitL := L#2000;
   A_3225_BTE06.Par.ParLimitH := L#8000;
   A_3225_BTE06.Par.ParLimitHH := L#10000;
   A_3225_BTE06.Par.ParMonTimeLL := 0;
   A_3225_BTE06.Par.ParMonTimeL := 0;
   A_3225_BTE06.Par.ParMonTimeMid := 0;
   A_3225_BTE06.Par.ParMonTimeH := 600;
   A_3225_BTE06.Par.ParMonTimeHH := 0;
   A_3225_BTE06.Par.ParDelayTimeDown := 10;
   A_3225_BTE06.Par.ParDelayTimeUp := 10;
   A_3225_BTE06.Par.ParDelayTime := 30;
   A_3225_BTE06.Par.OutMonTimeLL := 0;
   A_3225_BTE06.Par.OutMonTimeL := 0;
   A_3225_BTE06.Par.OutMonTimeMid := 0;
   A_3225_BTE06.Par.OutMonTimeH := 0;
   A_3225_BTE06.Par.OutMonTimeHH := 0;
   A_3225_BTE06.Par.OutDelayTimeDown := 0;
   A_3225_BTE06.Par.OutDelayTimeUp := 0;
   A_3225_BTE06.Par.OutDelayTime := 0;
   A_3225_BTE06.Par.Spare66 := 0;
   spare412[412] := B#16#0;
   spare412[413] := B#16#0;
   spare412[414] := B#16#0;
   spare412[415] := B#16#0;
   spare412[416] := B#16#0;
   spare412[417] := B#16#0;
   spare412[418] := B#16#0;
   spare412[419] := B#16#0;
   spare412[420] := B#16#0;
   spare412[421] := B#16#0;
   spare412[422] := B#16#0;
   spare412[423] := B#16#0;
   spare412[424] := B#16#0;
   spare412[425] := B#16#0;
   spare412[426] := B#16#0;
   spare412[427] := B#16#0;
   spare412[428] := B#16#0;
   spare412[429] := B#16#0;
   spare412[430] := B#16#0;
   spare412[431] := B#16#0;
   spare412[432] := B#16#0;
   spare412[433] := B#16#0;
   spare412[434] := B#16#0;
   spare412[435] := B#16#0;
   spare412[436] := B#16#0;
   spare412[437] := B#16#0;
   spare412[438] := B#16#0;
   spare412[439] := B#16#0;
   spare412[440] := B#16#0;
   spare412[441] := B#16#0;
   spare412[442] := B#16#0;
   spare412[443] := B#16#0;
   spare412[444] := B#16#0;
   spare412[445] := B#16#0;
   A_3225_MXZ01MA.Ma.StCode := 0;
   A_3225_MXZ01MA.Ma.InEnableRev := FALSE;
   A_3225_MXZ01MA.Ma.InEnableFwd := FALSE;
   A_3225_MXZ01MA.Ma.InOverrideHLOutlet := FALSE;
   A_3225_MXZ01MA.Ma.spare0203 := FALSE;
   A_3225_MXZ01MA.Ma.OutEdgeFaultReset := FALSE;
   A_3225_MXZ01MA.Ma.OutFaultResetFcttst := FALSE;
   A_3225_MXZ01MA.Ma.InpControlEBM := FALSE;
   A_3225_MXZ01MA.Ma.InpLocked := FALSE;
   A_3225_MXZ01MA.Ma.CmdOff := FALSE;
   A_3225_MXZ01MA.Ma.CmdOn := FALSE;
   A_3225_MXZ01MA.Ma.CmdNext := FALSE;
   A_3225_MXZ01MA.Ma.CmdFaultReset := FALSE;
   A_3225_MXZ01MA.Ma.InLocal := FALSE;
   A_3225_MXZ01MA.Ma.InManual := FALSE;
   A_3225_MXZ01MA.Ma.CmdTestEBM := FALSE;
   A_3225_MXZ01MA.Ma.InSeqStop := FALSE;
   A_3225_MXZ01MA.Ma.OutWarning := FALSE;
   A_3225_MXZ01MA.Ma.InfBMTopOk := FALSE;
   A_3225_MXZ01MA.Ma.InfBMBottomOk := FALSE;
   A_3225_MXZ01MA.Ma.InfSMOk := FALSE;
   A_3225_MXZ01MA.Ma.OutpFcttst_BM_Top := FALSE;
   A_3225_MXZ01MA.Ma.OutpFcttst_BM_Bottom := FALSE;
   A_3225_MXZ01MA.Ma.OutpFcttst_SM := FALSE;
   A_3225_MXZ01MA.Ma.OutpFaultReset := FALSE;
   A_3225_MXZ01MA.Ma.StStopped := FALSE;
   A_3225_MXZ01MA.Ma.StStarting := FALSE;
   A_3225_MXZ01MA.Ma.StStartedFwd := FALSE;
   A_3225_MXZ01MA.Ma.StStopping := FALSE;
   A_3225_MXZ01MA.Ma.StFault := FALSE;
   A_3225_MXZ01MA.Ma.StStartedRev := FALSE;
   A_3225_MXZ01MA.Ma.StLocked := FALSE;
   A_3225_MXZ01MA.Ma.OutTestTime := 0;
   A_3225_MXZ01MA.Ma.Par.ParObjectNo := 29706;
   A_3225_MXZ01MA.Ma.Par.ParWithMon1 := TRUE;
   A_3225_MXZ01MA.Ma.Par.ParWithMon3 := FALSE;
   A_3225_MXZ01MA.Ma.Par.ParWithMon4 := FALSE;
   A_3225_MXZ01MA.Ma.Par.ParWithMon5 := FALSE;
   A_3225_MXZ01MA.Ma.Par.ParWithMon6 := FALSE;
   A_3225_MXZ01MA.Ma.Par.ParMon1IsHL := FALSE;
   A_3225_MXZ01MA.Ma.Par.ParMon1IsLS := TRUE;
   A_3225_MXZ01MA.Ma.Par.ParMon1StopByFault := TRUE;
   A_3225_MXZ01MA.Ma.Par.ParMon2IsLS := FALSE;
   A_3225_MXZ01MA.Ma.Par.ParMon3IsLS := FALSE;
   A_3225_MXZ01MA.Ma.Par.ParMon4AsWarning := FALSE;
   A_3225_MXZ01MA.Ma.Par.ParMon4StopByFault := FALSE;
   A_3225_MXZ01MA.Ma.Par.ParMon4IsLS := FALSE;
   A_3225_MXZ01MA.Ma.Par.ParEBM := FALSE;
   A_3225_MXZ01MA.Ma.Par.ParMon4IsSM := FALSE;
   A_3225_MXZ01MA.A_3225_KCU04.StCode := 0;
   A_3225_MXZ01MA.A_3225_KCU04.InMonTrue := FALSE;
   A_3225_MXZ01MA.A_3225_KCU04.InMonFalse := FALSE;
   A_3225_MXZ01MA.A_3225_KCU04.InPreAlarmTrue := FALSE;
   A_3225_MXZ01MA.A_3225_KCU04.InPreAlarmFalse := FALSE;
   A_3225_MXZ01MA.A_3225_KCU04.InStopTrueTime := FALSE;
   A_3225_MXZ01MA.A_3225_KCU04.InStopFalseTime := FALSE;
   A_3225_MXZ01MA.A_3225_KCU04.InpTrue := FALSE;
   A_3225_MXZ01MA.A_3225_KCU04.InpFaultDev := FALSE;
   A_3225_MXZ01MA.A_3225_KCU04.CmdRstTrueTime := FALSE;
   A_3225_MXZ01MA.A_3225_KCU04.CmdRstFalseTime := FALSE;
   A_3225_MXZ01MA.A_3225_KCU04.CmdRunTimeoutTime := FALSE;
   A_3225_MXZ01MA.A_3225_KCU04.CmdFaultReset := FALSE;
   A_3225_MXZ01MA.A_3225_KCU04.InLocal := FALSE;
   A_3225_MXZ01MA.A_3225_KCU04.spare0305 := FALSE;
   A_3225_MXZ01MA.A_3225_KCU04.InReport := FALSE;
   A_3225_MXZ01MA.A_3225_KCU04.OutTimeoutTime := FALSE;
   A_3225_MXZ01MA.A_3225_KCU04.InHWStop := FALSE;
   A_3225_MXZ01MA.A_3225_KCU04.InDPFault := FALSE;
   A_3225_MXZ01MA.A_3225_KCU04.OutPreAlarmTrue := FALSE;
   A_3225_MXZ01MA.A_3225_KCU04.OutPreAlarmFalse := FALSE;
   A_3225_MXZ01MA.A_3225_KCU04.OutFlagPos := FALSE;
   A_3225_MXZ01MA.A_3225_KCU04.OutFlagNeg := FALSE;
   A_3225_MXZ01MA.A_3225_KCU04.OutpFaultReset := FALSE;
   A_3225_MXZ01MA.A_3225_KCU04.OutTrue := FALSE;
   A_3225_MXZ01MA.A_3225_KCU04.StFalse := FALSE;
   A_3225_MXZ01MA.A_3225_KCU04.StCtoTrue := FALSE;
   A_3225_MXZ01MA.A_3225_KCU04.StTrue := FALSE;
   A_3225_MXZ01MA.A_3225_KCU04.StCtoFalse := FALSE;
   A_3225_MXZ01MA.A_3225_KCU04.StFault := FALSE;
   A_3225_MXZ01MA.A_3225_KCU04.OutAlarmNrLog := 0;
   A_3225_MXZ01MA.A_3225_KCU04.Par.ParObjectNo := 29707;
   A_3225_MXZ01MA.A_3225_KCU04.Par.ParMsgType := 7154;
   A_3225_MXZ01MA.A_3225_KCU04.Par.ParHornCode := 11;
   A_3225_MXZ01MA.A_3225_KCU04.Par.ParLogOff := FALSE;
   A_3225_MXZ01MA.A_3225_KCU04.Par.spare0401 := FALSE;
   A_3225_MXZ01MA.A_3225_KCU04.Par.Par2WorkingCond := FALSE;
   A_3225_MXZ01MA.A_3225_KCU04.Par.ParFaultRetry := FALSE;
   A_3225_MXZ01MA.A_3225_KCU04.Par.ParBinLevel := FALSE;
   A_3225_MXZ01MA.A_3225_KCU04.Par.ParDelayChange := 20;
   A_3225_MXZ01MA.A_3225_KCU04.Par.ParDelayTrue := 10;
   A_3225_MXZ01MA.A_3225_KCU04.Par.ParDelayFalse := 0;
   A_3225_MXZ01MA.A_3225_KCU04.Par.ParTimeoutTrue := 0;
   A_3225_MXZ01MA.A_3225_KCU04.Par.ParTimeoutFalse := 0;
   A_3225_MXZ01MA.A_3225_KCU04.Par.OutMonTime := 0;
   A_3225_MXZ01MA.A_3225_KCU04.Par.OutTransitionTime := 0;
   A_3225_MXZ01MA.A_3225_KCU04.Par.OutMonTrue := FALSE;
   A_3225_MXZ01MA.A_3225_KCU04.Par.OutMonFalse := FALSE;
   A_3225_MXZ01MA.A_3225_KCU04.Par.OutFlagFaultDev := FALSE;
   A_3225_MXZ01MA.A_3225_KCU04.Par.OutDelayTime := 0;
   A_3225_MXZ01MA.A_3225_MXZ01_SM.StCode := 0;
   A_3225_MXZ01MA.A_3225_MXZ01_SM.InMonTrue := FALSE;
   A_3225_MXZ01MA.A_3225_MXZ01_SM.InMonFalse := FALSE;
   A_3225_MXZ01MA.A_3225_MXZ01_SM.InPreAlarmTrue := FALSE;
   A_3225_MXZ01MA.A_3225_MXZ01_SM.InPreAlarmFalse := FALSE;
   A_3225_MXZ01MA.A_3225_MXZ01_SM.InStopTrueTime := FALSE;
   A_3225_MXZ01MA.A_3225_MXZ01_SM.InStopFalseTime := FALSE;
   A_3225_MXZ01MA.A_3225_MXZ01_SM.InpTrue := FALSE;
   A_3225_MXZ01MA.A_3225_MXZ01_SM.InpFaultDev := FALSE;
   A_3225_MXZ01MA.A_3225_MXZ01_SM.CmdRstTrueTime := FALSE;
   A_3225_MXZ01MA.A_3225_MXZ01_SM.CmdRstFalseTime := FALSE;
   A_3225_MXZ01MA.A_3225_MXZ01_SM.CmdRunTimeoutTime := FALSE;
   A_3225_MXZ01MA.A_3225_MXZ01_SM.CmdFaultReset := FALSE;
   A_3225_MXZ01MA.A_3225_MXZ01_SM.InLocal := FALSE;
   A_3225_MXZ01MA.A_3225_MXZ01_SM.spare0305 := FALSE;
   A_3225_MXZ01MA.A_3225_MXZ01_SM.InReport := FALSE;
   A_3225_MXZ01MA.A_3225_MXZ01_SM.OutTimeoutTime := FALSE;
   A_3225_MXZ01MA.A_3225_MXZ01_SM.InHWStop := FALSE;
   A_3225_MXZ01MA.A_3225_MXZ01_SM.InDPFault := FALSE;
   A_3225_MXZ01MA.A_3225_MXZ01_SM.OutPreAlarmTrue := FALSE;
   A_3225_MXZ01MA.A_3225_MXZ01_SM.OutPreAlarmFalse := FALSE;
   A_3225_MXZ01MA.A_3225_MXZ01_SM.OutFlagPos := FALSE;
   A_3225_MXZ01MA.A_3225_MXZ01_SM.OutFlagNeg := FALSE;
   A_3225_MXZ01MA.A_3225_MXZ01_SM.OutpFaultReset := FALSE;
   A_3225_MXZ01MA.A_3225_MXZ01_SM.OutTrue := FALSE;
   A_3225_MXZ01MA.A_3225_MXZ01_SM.StFalse := FALSE;
   A_3225_MXZ01MA.A_3225_MXZ01_SM.StCtoTrue := FALSE;
   A_3225_MXZ01MA.A_3225_MXZ01_SM.StTrue := FALSE;
   A_3225_MXZ01MA.A_3225_MXZ01_SM.StCtoFalse := FALSE;
   A_3225_MXZ01MA.A_3225_MXZ01_SM.StFault := FALSE;
   A_3225_MXZ01MA.A_3225_MXZ01_SM.OutAlarmNrLog := 0;
   A_3225_MXZ01MA.A_3225_MXZ01_SM.Par.ParObjectNo := 29708;
   A_3225_MXZ01MA.A_3225_MXZ01_SM.Par.ParMsgType := 7135;
   A_3225_MXZ01MA.A_3225_MXZ01_SM.Par.ParHornCode := 11;
   A_3225_MXZ01MA.A_3225_MXZ01_SM.Par.ParLogOff := FALSE;
   A_3225_MXZ01MA.A_3225_MXZ01_SM.Par.spare0401 := FALSE;
   A_3225_MXZ01MA.A_3225_MXZ01_SM.Par.Par2WorkingCond := TRUE;
   A_3225_MXZ01MA.A_3225_MXZ01_SM.Par.ParFaultRetry := FALSE;
   A_3225_MXZ01MA.A_3225_MXZ01_SM.Par.ParBinLevel := FALSE;
   A_3225_MXZ01MA.A_3225_MXZ01_SM.Par.ParDelayChange := 0;
   A_3225_MXZ01MA.A_3225_MXZ01_SM.Par.ParDelayTrue := 10;
   A_3225_MXZ01MA.A_3225_MXZ01_SM.Par.ParDelayFalse := 0;
   A_3225_MXZ01MA.A_3225_MXZ01_SM.Par.ParTimeoutTrue := 50;
   A_3225_MXZ01MA.A_3225_MXZ01_SM.Par.ParTimeoutFalse := 0;
   A_3225_MXZ01MA.A_3225_MXZ01_SM.Par.OutMonTime := 0;
   A_3225_MXZ01MA.A_3225_MXZ01_SM.Par.OutTransitionTime := 0;
   A_3225_MXZ01MA.A_3225_MXZ01_SM.Par.OutMonTrue := FALSE;
   A_3225_MXZ01MA.A_3225_MXZ01_SM.Par.OutMonFalse := FALSE;
   A_3225_MXZ01MA.A_3225_MXZ01_SM.Par.OutFlagFaultDev := FALSE;
   A_3225_MXZ01MA.A_3225_MXZ01_SM.Par.OutDelayTime := 0;
   A_3225_MXZ01MA.Mon3.StCode := 0;
   A_3225_MXZ01MA.Mon3.InMonTrue := FALSE;
   A_3225_MXZ01MA.Mon3.InMonFalse := FALSE;
   A_3225_MXZ01MA.Mon3.InPreAlarmTrue := FALSE;
   A_3225_MXZ01MA.Mon3.InPreAlarmFalse := FALSE;
   A_3225_MXZ01MA.Mon3.InStopTrueTime := FALSE;
   A_3225_MXZ01MA.Mon3.InStopFalseTime := FALSE;
   A_3225_MXZ01MA.Mon3.InpTrue := FALSE;
   A_3225_MXZ01MA.Mon3.InpFaultDev := FALSE;
   A_3225_MXZ01MA.Mon3.CmdRstTrueTime := FALSE;
   A_3225_MXZ01MA.Mon3.CmdRstFalseTime := FALSE;
   A_3225_MXZ01MA.Mon3.CmdRunTimeoutTime := FALSE;
   A_3225_MXZ01MA.Mon3.CmdFaultReset := FALSE;
   A_3225_MXZ01MA.Mon3.InLocal := FALSE;
   A_3225_MXZ01MA.Mon3.spare0305 := FALSE;
   A_3225_MXZ01MA.Mon3.InReport := FALSE;
   A_3225_MXZ01MA.Mon3.OutTimeoutTime := FALSE;
   A_3225_MXZ01MA.Mon3.InHWStop := FALSE;
   A_3225_MXZ01MA.Mon3.InDPFault := FALSE;
   A_3225_MXZ01MA.Mon3.OutPreAlarmTrue := FALSE;
   A_3225_MXZ01MA.Mon3.OutPreAlarmFalse := FALSE;
   A_3225_MXZ01MA.Mon3.OutFlagPos := FALSE;
   A_3225_MXZ01MA.Mon3.OutFlagNeg := FALSE;
   A_3225_MXZ01MA.Mon3.OutpFaultReset := FALSE;
   A_3225_MXZ01MA.Mon3.OutTrue := FALSE;
   A_3225_MXZ01MA.Mon3.StFalse := FALSE;
   A_3225_MXZ01MA.Mon3.StCtoTrue := FALSE;
   A_3225_MXZ01MA.Mon3.StTrue := FALSE;
   A_3225_MXZ01MA.Mon3.StCtoFalse := FALSE;
   A_3225_MXZ01MA.Mon3.StFault := FALSE;
   A_3225_MXZ01MA.Mon3.OutAlarmNrLog := 0;
   A_3225_MXZ01MA.Mon3.Par.ParObjectNo := 0;
   A_3225_MXZ01MA.Mon3.Par.ParMsgType := 0;
   A_3225_MXZ01MA.Mon3.Par.ParHornCode := 0;
   A_3225_MXZ01MA.Mon3.Par.ParLogOff := FALSE;
   A_3225_MXZ01MA.Mon3.Par.spare0401 := FALSE;
   A_3225_MXZ01MA.Mon3.Par.Par2WorkingCond := FALSE;
   A_3225_MXZ01MA.Mon3.Par.ParFaultRetry := FALSE;
   A_3225_MXZ01MA.Mon3.Par.ParBinLevel := FALSE;
   A_3225_MXZ01MA.Mon3.Par.ParDelayChange := 0;
   A_3225_MXZ01MA.Mon3.Par.ParDelayTrue := 0;
   A_3225_MXZ01MA.Mon3.Par.ParDelayFalse := 0;
   A_3225_MXZ01MA.Mon3.Par.ParTimeoutTrue := 0;
   A_3225_MXZ01MA.Mon3.Par.ParTimeoutFalse := 0;
   A_3225_MXZ01MA.Mon3.Par.OutMonTime := 0;
   A_3225_MXZ01MA.Mon3.Par.OutTransitionTime := 0;
   A_3225_MXZ01MA.Mon3.Par.OutMonTrue := FALSE;
   A_3225_MXZ01MA.Mon3.Par.OutMonFalse := FALSE;
   A_3225_MXZ01MA.Mon3.Par.OutFlagFaultDev := FALSE;
   A_3225_MXZ01MA.Mon3.Par.OutDelayTime := 0;
   A_3225_MXZ01MA.Mon4.StCode := 0;
   A_3225_MXZ01MA.Mon4.InMonTrue := FALSE;
   A_3225_MXZ01MA.Mon4.InMonFalse := FALSE;
   A_3225_MXZ01MA.Mon4.InPreAlarmTrue := FALSE;
   A_3225_MXZ01MA.Mon4.InPreAlarmFalse := FALSE;
   A_3225_MXZ01MA.Mon4.InStopTrueTime := FALSE;
   A_3225_MXZ01MA.Mon4.InStopFalseTime := FALSE;
   A_3225_MXZ01MA.Mon4.InpTrue := FALSE;
   A_3225_MXZ01MA.Mon4.InpFaultDev := FALSE;
   A_3225_MXZ01MA.Mon4.CmdRstTrueTime := FALSE;
   A_3225_MXZ01MA.Mon4.CmdRstFalseTime := FALSE;
   A_3225_MXZ01MA.Mon4.CmdRunTimeoutTime := FALSE;
   A_3225_MXZ01MA.Mon4.CmdFaultReset := FALSE;
   A_3225_MXZ01MA.Mon4.InLocal := FALSE;
   A_3225_MXZ01MA.Mon4.spare0305 := FALSE;
   A_3225_MXZ01MA.Mon4.InReport := FALSE;
   A_3225_MXZ01MA.Mon4.OutTimeoutTime := FALSE;
   A_3225_MXZ01MA.Mon4.InHWStop := FALSE;
   A_3225_MXZ01MA.Mon4.InDPFault := FALSE;
   A_3225_MXZ01MA.Mon4.OutPreAlarmTrue := FALSE;
   A_3225_MXZ01MA.Mon4.OutPreAlarmFalse := FALSE;
   A_3225_MXZ01MA.Mon4.OutFlagPos := FALSE;
   A_3225_MXZ01MA.Mon4.OutFlagNeg := FALSE;
   A_3225_MXZ01MA.Mon4.OutpFaultReset := FALSE;
   A_3225_MXZ01MA.Mon4.OutTrue := FALSE;
   A_3225_MXZ01MA.Mon4.StFalse := FALSE;
   A_3225_MXZ01MA.Mon4.StCtoTrue := FALSE;
   A_3225_MXZ01MA.Mon4.StTrue := FALSE;
   A_3225_MXZ01MA.Mon4.StCtoFalse := FALSE;
   A_3225_MXZ01MA.Mon4.StFault := FALSE;
   A_3225_MXZ01MA.Mon4.OutAlarmNrLog := 0;
   A_3225_MXZ01MA.Mon4.Par.ParObjectNo := 0;
   A_3225_MXZ01MA.Mon4.Par.ParMsgType := 0;
   A_3225_MXZ01MA.Mon4.Par.ParHornCode := 0;
   A_3225_MXZ01MA.Mon4.Par.ParLogOff := FALSE;
   A_3225_MXZ01MA.Mon4.Par.spare0401 := FALSE;
   A_3225_MXZ01MA.Mon4.Par.Par2WorkingCond := FALSE;
   A_3225_MXZ01MA.Mon4.Par.ParFaultRetry := FALSE;
   A_3225_MXZ01MA.Mon4.Par.ParBinLevel := FALSE;
   A_3225_MXZ01MA.Mon4.Par.ParDelayChange := 0;
   A_3225_MXZ01MA.Mon4.Par.ParDelayTrue := 0;
   A_3225_MXZ01MA.Mon4.Par.ParDelayFalse := 0;
   A_3225_MXZ01MA.Mon4.Par.ParTimeoutTrue := 0;
   A_3225_MXZ01MA.Mon4.Par.ParTimeoutFalse := 0;
   A_3225_MXZ01MA.Mon4.Par.OutMonTime := 0;
   A_3225_MXZ01MA.Mon4.Par.OutTransitionTime := 0;
   A_3225_MXZ01MA.Mon4.Par.OutMonTrue := FALSE;
   A_3225_MXZ01MA.Mon4.Par.OutMonFalse := FALSE;
   A_3225_MXZ01MA.Mon4.Par.OutFlagFaultDev := FALSE;
   A_3225_MXZ01MA.Mon4.Par.OutDelayTime := 0;
   A_3225_MXZ01MA.Mon5.StCode := 0;
   A_3225_MXZ01MA.Mon5.InMonTrue := FALSE;
   A_3225_MXZ01MA.Mon5.InMonFalse := FALSE;
   A_3225_MXZ01MA.Mon5.InPreAlarmTrue := FALSE;
   A_3225_MXZ01MA.Mon5.InPreAlarmFalse := FALSE;
   A_3225_MXZ01MA.Mon5.InStopTrueTime := FALSE;
   A_3225_MXZ01MA.Mon5.InStopFalseTime := FALSE;
   A_3225_MXZ01MA.Mon5.InpTrue := FALSE;
   A_3225_MXZ01MA.Mon5.InpFaultDev := FALSE;
   A_3225_MXZ01MA.Mon5.CmdRstTrueTime := FALSE;
   A_3225_MXZ01MA.Mon5.CmdRstFalseTime := FALSE;
   A_3225_MXZ01MA.Mon5.CmdRunTimeoutTime := FALSE;
   A_3225_MXZ01MA.Mon5.CmdFaultReset := FALSE;
   A_3225_MXZ01MA.Mon5.InLocal := FALSE;
   A_3225_MXZ01MA.Mon5.spare0305 := FALSE;
   A_3225_MXZ01MA.Mon5.InReport := FALSE;
   A_3225_MXZ01MA.Mon5.OutTimeoutTime := FALSE;
   A_3225_MXZ01MA.Mon5.InHWStop := FALSE;
   A_3225_MXZ01MA.Mon5.InDPFault := FALSE;
   A_3225_MXZ01MA.Mon5.OutPreAlarmTrue := FALSE;
   A_3225_MXZ01MA.Mon5.OutPreAlarmFalse := FALSE;
   A_3225_MXZ01MA.Mon5.OutFlagPos := FALSE;
   A_3225_MXZ01MA.Mon5.OutFlagNeg := FALSE;
   A_3225_MXZ01MA.Mon5.OutpFaultReset := FALSE;
   A_3225_MXZ01MA.Mon5.OutTrue := FALSE;
   A_3225_MXZ01MA.Mon5.StFalse := FALSE;
   A_3225_MXZ01MA.Mon5.StCtoTrue := FALSE;
   A_3225_MXZ01MA.Mon5.StTrue := FALSE;
   A_3225_MXZ01MA.Mon5.StCtoFalse := FALSE;
   A_3225_MXZ01MA.Mon5.StFault := FALSE;
   A_3225_MXZ01MA.Mon5.OutAlarmNrLog := 0;
   A_3225_MXZ01MA.Mon5.Par.ParObjectNo := 0;
   A_3225_MXZ01MA.Mon5.Par.ParMsgType := 0;
   A_3225_MXZ01MA.Mon5.Par.ParHornCode := 0;
   A_3225_MXZ01MA.Mon5.Par.ParLogOff := FALSE;
   A_3225_MXZ01MA.Mon5.Par.spare0401 := FALSE;
   A_3225_MXZ01MA.Mon5.Par.Par2WorkingCond := FALSE;
   A_3225_MXZ01MA.Mon5.Par.ParFaultRetry := FALSE;
   A_3225_MXZ01MA.Mon5.Par.ParBinLevel := FALSE;
   A_3225_MXZ01MA.Mon5.Par.ParDelayChange := 0;
   A_3225_MXZ01MA.Mon5.Par.ParDelayTrue := 0;
   A_3225_MXZ01MA.Mon5.Par.ParDelayFalse := 0;
   A_3225_MXZ01MA.Mon5.Par.ParTimeoutTrue := 0;
   A_3225_MXZ01MA.Mon5.Par.ParTimeoutFalse := 0;
   A_3225_MXZ01MA.Mon5.Par.OutMonTime := 0;
   A_3225_MXZ01MA.Mon5.Par.OutTransitionTime := 0;
   A_3225_MXZ01MA.Mon5.Par.OutMonTrue := FALSE;
   A_3225_MXZ01MA.Mon5.Par.OutMonFalse := FALSE;
   A_3225_MXZ01MA.Mon5.Par.OutFlagFaultDev := FALSE;
   A_3225_MXZ01MA.Mon5.Par.OutDelayTime := 0;
   A_3225_MXZ01MA.Mon6.StCode := 0;
   A_3225_MXZ01MA.Mon6.InMonTrue := FALSE;
   A_3225_MXZ01MA.Mon6.InMonFalse := FALSE;
   A_3225_MXZ01MA.Mon6.InPreAlarmTrue := FALSE;
   A_3225_MXZ01MA.Mon6.InPreAlarmFalse := FALSE;
   A_3225_MXZ01MA.Mon6.InStopTrueTime := FALSE;
   A_3225_MXZ01MA.Mon6.InStopFalseTime := FALSE;
   A_3225_MXZ01MA.Mon6.InpTrue := FALSE;
   A_3225_MXZ01MA.Mon6.InpFaultDev := FALSE;
   A_3225_MXZ01MA.Mon6.CmdRstTrueTime := FALSE;
   A_3225_MXZ01MA.Mon6.CmdRstFalseTime := FALSE;
   A_3225_MXZ01MA.Mon6.CmdRunTimeoutTime := FALSE;
   A_3225_MXZ01MA.Mon6.CmdFaultReset := FALSE;
   A_3225_MXZ01MA.Mon6.InLocal := FALSE;
   A_3225_MXZ01MA.Mon6.spare0305 := FALSE;
   A_3225_MXZ01MA.Mon6.InReport := FALSE;
   A_3225_MXZ01MA.Mon6.OutTimeoutTime := FALSE;
   A_3225_MXZ01MA.Mon6.InHWStop := FALSE;
   A_3225_MXZ01MA.Mon6.InDPFault := FALSE;
   A_3225_MXZ01MA.Mon6.OutPreAlarmTrue := FALSE;
   A_3225_MXZ01MA.Mon6.OutPreAlarmFalse := FALSE;
   A_3225_MXZ01MA.Mon6.OutFlagPos := FALSE;
   A_3225_MXZ01MA.Mon6.OutFlagNeg := FALSE;
   A_3225_MXZ01MA.Mon6.OutpFaultReset := FALSE;
   A_3225_MXZ01MA.Mon6.OutTrue := FALSE;
   A_3225_MXZ01MA.Mon6.StFalse := FALSE;
   A_3225_MXZ01MA.Mon6.StCtoTrue := FALSE;
   A_3225_MXZ01MA.Mon6.StTrue := FALSE;
   A_3225_MXZ01MA.Mon6.StCtoFalse := FALSE;
   A_3225_MXZ01MA.Mon6.StFault := FALSE;
   A_3225_MXZ01MA.Mon6.OutAlarmNrLog := 0;
   A_3225_MXZ01MA.Mon6.Par.ParObjectNo := 0;
   A_3225_MXZ01MA.Mon6.Par.ParMsgType := 0;
   A_3225_MXZ01MA.Mon6.Par.ParHornCode := 0;
   A_3225_MXZ01MA.Mon6.Par.ParLogOff := FALSE;
   A_3225_MXZ01MA.Mon6.Par.spare0401 := FALSE;
   A_3225_MXZ01MA.Mon6.Par.Par2WorkingCond := FALSE;
   A_3225_MXZ01MA.Mon6.Par.ParFaultRetry := FALSE;
   A_3225_MXZ01MA.Mon6.Par.ParBinLevel := FALSE;
   A_3225_MXZ01MA.Mon6.Par.ParDelayChange := 0;
   A_3225_MXZ01MA.Mon6.Par.ParDelayTrue := 0;
   A_3225_MXZ01MA.Mon6.Par.ParDelayFalse := 0;
   A_3225_MXZ01MA.Mon6.Par.ParTimeoutTrue := 0;
   A_3225_MXZ01MA.Mon6.Par.ParTimeoutFalse := 0;
   A_3225_MXZ01MA.Mon6.Par.OutMonTime := 0;
   A_3225_MXZ01MA.Mon6.Par.OutTransitionTime := 0;
   A_3225_MXZ01MA.Mon6.Par.OutMonTrue := FALSE;
   A_3225_MXZ01MA.Mon6.Par.OutMonFalse := FALSE;
   A_3225_MXZ01MA.Mon6.Par.OutFlagFaultDev := FALSE;
   A_3225_MXZ01MA.Mon6.Par.OutDelayTime := 0;
   A_3225_MXZ01MA.A_3225_MXZ01.StCode := 0;
   A_3225_MXZ01MA.A_3225_MXZ01.InEnableRev := FALSE;
   A_3225_MXZ01MA.A_3225_MXZ01.InEnableFwd := FALSE;
   A_3225_MXZ01MA.A_3225_MXZ01.InSlow := FALSE;
   A_3225_MXZ01MA.A_3225_MXZ01.InpRunSlow := FALSE;
   A_3225_MXZ01MA.A_3225_MXZ01.InpRunFast := FALSE;
   A_3225_MXZ01MA.A_3225_MXZ01.InpRunRev := FALSE;
   A_3225_MXZ01MA.A_3225_MXZ01.InpRunFwd := FALSE;
   A_3225_MXZ01MA.A_3225_MXZ01.InpFaultDev := FALSE;
   A_3225_MXZ01MA.A_3225_MXZ01.CmdOff := FALSE;
   A_3225_MXZ01MA.A_3225_MXZ01.CmdOn := FALSE;
   A_3225_MXZ01MA.A_3225_MXZ01.CmdNext := FALSE;
   A_3225_MXZ01MA.A_3225_MXZ01.CmdFaultReset := FALSE;
   A_3225_MXZ01MA.A_3225_MXZ01.InLocal := FALSE;
   A_3225_MXZ01MA.A_3225_MXZ01.InManual := FALSE;
   A_3225_MXZ01MA.A_3225_MXZ01.InReport := FALSE;
   A_3225_MXZ01MA.A_3225_MXZ01.InSeqStop := FALSE;
   A_3225_MXZ01MA.A_3225_MXZ01.InHWStop := FALSE;
   A_3225_MXZ01MA.A_3225_MXZ01.InDPFault := FALSE;
   A_3225_MXZ01MA.A_3225_MXZ01.OutIdling := FALSE;
   A_3225_MXZ01MA.A_3225_MXZ01.OutpRunSlow := FALSE;
   A_3225_MXZ01MA.A_3225_MXZ01.OutpRunFast := FALSE;
   A_3225_MXZ01MA.A_3225_MXZ01.OutpRunRev := FALSE;
   A_3225_MXZ01MA.A_3225_MXZ01.OutpRunFwd := FALSE;
   A_3225_MXZ01MA.A_3225_MXZ01.OutpFaultReset := FALSE;
   A_3225_MXZ01MA.A_3225_MXZ01.StStopped := FALSE;
   A_3225_MXZ01MA.A_3225_MXZ01.StStarting := FALSE;
   A_3225_MXZ01MA.A_3225_MXZ01.StStartedFwd := FALSE;
   A_3225_MXZ01MA.A_3225_MXZ01.StStopping := FALSE;
   A_3225_MXZ01MA.A_3225_MXZ01.StFault := FALSE;
   A_3225_MXZ01MA.A_3225_MXZ01.StStartedRev := FALSE;
   A_3225_MXZ01MA.A_3225_MXZ01.InOutManSlow := FALSE;
   A_3225_MXZ01MA.A_3225_MXZ01.InOutManRev := FALSE;
   A_3225_MXZ01MA.A_3225_MXZ01.OutAlarmNrLog := 0;
   A_3225_MXZ01MA.A_3225_MXZ01.Par.ParObjectNo := 29709;
   A_3225_MXZ01MA.A_3225_MXZ01.Par.ParMsgType := 7053;
   A_3225_MXZ01MA.A_3225_MXZ01.Par.ParHornCode := 11;
   A_3225_MXZ01MA.A_3225_MXZ01.Par.ParLogOff := FALSE;
   A_3225_MXZ01MA.A_3225_MXZ01.Par.ParManual := TRUE;
   A_3225_MXZ01MA.A_3225_MXZ01.Par.ParRestartDelay := FALSE;
   A_3225_MXZ01MA.A_3225_MXZ01.Par.Par2Speed := FALSE;
   A_3225_MXZ01MA.A_3225_MXZ01.Par.ParHeavyStartup := FALSE;
   A_3225_MXZ01MA.A_3225_MXZ01.Par.spare45 := FALSE;
   A_3225_MXZ01MA.A_3225_MXZ01.Par.spare46 := FALSE;
   A_3225_MXZ01MA.A_3225_MXZ01.Par.OutEdgeFaultReset := FALSE;
   A_3225_MXZ01MA.A_3225_MXZ01.Par.OutDelayFault := FALSE;
   A_3225_MXZ01MA.A_3225_MXZ01.Par.OutFlagFaultDev := FALSE;
   A_3225_MXZ01MA.A_3225_MXZ01.Par.ParMonTime := 20;
   A_3225_MXZ01MA.A_3225_MXZ01.Par.ParStartingTime := 20;
   A_3225_MXZ01MA.A_3225_MXZ01.Par.ParStoppingTime := 0;
   A_3225_MXZ01MA.A_3225_MXZ01.Par.ParIdlingTime := 0;
   A_3225_MXZ01MA.A_3225_MXZ01.Par.ParDelayTime := 10;
   A_3225_MXZ01MA.A_3225_MXZ01.Par.OutMonTime := 0;
   A_3225_MXZ01MA.A_3225_MXZ01.Par.OutTransitionTime := 0;
   A_3225_MXZ01MA.A_3225_MXZ01.Par.OutDelayTime := 0;
   A_3225_MXZ01MA.A_3225_MXZ01.Par.InOutManPulseLen := 0;
   A_3225_TSC01_AC.StCode := 0;
   A_3225_TSC01_AC.InMonLL := FALSE;
   A_3225_TSC01_AC.InMonL := FALSE;
   A_3225_TSC01_AC.InMonMid := FALSE;
   A_3225_TSC01_AC.InMonH := FALSE;
   A_3225_TSC01_AC.InMonHH := FALSE;
   A_3225_TSC01_AC.spare0205 := FALSE;
   A_3225_TSC01_AC.InpFaultAI := FALSE;
   A_3225_TSC01_AC.InpFaultDev := FALSE;
   A_3225_TSC01_AC.InHWStop := FALSE;
   A_3225_TSC01_AC.InDPFault := FALSE;
   A_3225_TSC01_AC.InDisable := FALSE;
   A_3225_TSC01_AC.CmdFaultReset := FALSE;
   A_3225_TSC01_AC.InLocal := FALSE;
   A_3225_TSC01_AC.spare0305 := FALSE;
   A_3225_TSC01_AC.InReport := FALSE;
   A_3225_TSC01_AC.spare0307 := FALSE;
   A_3225_TSC01_AC.OutLL := FALSE;
   A_3225_TSC01_AC.OutL := FALSE;
   A_3225_TSC01_AC.OutH := FALSE;
   A_3225_TSC01_AC.OutHH := FALSE;
   A_3225_TSC01_AC.OutOverflow := FALSE;
   A_3225_TSC01_AC.spare0405 := FALSE;
   A_3225_TSC01_AC.OutFaultAI := FALSE;
   A_3225_TSC01_AC.spare0407 := FALSE;
   A_3225_TSC01_AC.StLL := FALSE;
   A_3225_TSC01_AC.StL := FALSE;
   A_3225_TSC01_AC.StMid := FALSE;
   A_3225_TSC01_AC.StH := FALSE;
   A_3225_TSC01_AC.StHH := FALSE;
   A_3225_TSC01_AC.StFaultAI := FALSE;
   A_3225_TSC01_AC.OutWarning := FALSE;
   A_3225_TSC01_AC.OutFaulted := FALSE;
   A_3225_TSC01_AC.InpValue := 0;
   A_3225_TSC01_AC.OutValuePc := 0;
   A_3225_TSC01_AC.OutValueUnits := L#0;
   A_3225_TSC01_AC.Msg.WarningDoneLL := FALSE;
   A_3225_TSC01_AC.Msg.WarningDoneL := FALSE;
   A_3225_TSC01_AC.Msg.WarningDoneMid := FALSE;
   A_3225_TSC01_AC.Msg.WarningDoneH := FALSE;
   A_3225_TSC01_AC.Msg.WarningDoneHH := FALSE;
   A_3225_TSC01_AC.Msg.FaultDoneLL := FALSE;
   A_3225_TSC01_AC.Msg.FaultDoneL := FALSE;
   A_3225_TSC01_AC.Msg.FaultDoneMid := FALSE;
   A_3225_TSC01_AC.Msg.FaultDoneH := FALSE;
   A_3225_TSC01_AC.Msg.FaultDoneHH := FALSE;
   A_3225_TSC01_AC.Msg.FaultDoneDev := FALSE;
   A_3225_TSC01_AC.Msg.FaultDoneAI := FALSE;
   A_3225_TSC01_AC.OutAlarmNrLog := 0;
   A_3225_TSC01_AC.Par.ParObjectNo := 29710;
   A_3225_TSC01_AC.Par.ParMsgType := 7252;
   A_3225_TSC01_AC.Par.ParHornCode := 11;
   A_3225_TSC01_AC.Par.ParLogOff := FALSE;
   A_3225_TSC01_AC.Par.ParSpare0401 := FALSE;
   A_3225_TSC01_AC.Par.ParValueByUser := FALSE;
   A_3225_TSC01_AC.Par.ParLimitsPc := TRUE;
   A_3225_TSC01_AC.Par.ParWago := FALSE;
   A_3225_TSC01_AC.Par.ParNoHornByWarning := FALSE;
   A_3225_TSC01_AC.Par.ParWarningLL := FALSE;
   A_3225_TSC01_AC.Par.ParWarningL := FALSE;
   A_3225_TSC01_AC.Par.ParWarningMid := FALSE;
   A_3225_TSC01_AC.Par.ParWarningH := FALSE;
   A_3225_TSC01_AC.Par.ParWarningHH := FALSE;
   A_3225_TSC01_AC.Par.ParPreAlarmLL := FALSE;
   A_3225_TSC01_AC.Par.ParPreAlarmL := FALSE;
   A_3225_TSC01_AC.Par.ParPreAlarmMid := FALSE;
   A_3225_TSC01_AC.Par.ParPreAlarmH := FALSE;
   A_3225_TSC01_AC.Par.ParPreAlarmHH := FALSE;
   A_3225_TSC01_AC.Par.ParUnitsByZeroDigit := L#0;
   A_3225_TSC01_AC.Par.ParUnitsByMaxDigit := L#25384;
   A_3225_TSC01_AC.Par.ParUnitsBy100Pc := L#10000;
   A_3225_TSC01_AC.Par.ParLimitLL := L#-1;
   A_3225_TSC01_AC.Par.ParLimitL := L#0;
   A_3225_TSC01_AC.Par.ParLimitH := L#5400;
   A_3225_TSC01_AC.Par.ParLimitHH := L#6000;
   A_3225_TSC01_AC.Par.ParMonTimeLL := 0;
   A_3225_TSC01_AC.Par.ParMonTimeL := 0;
   A_3225_TSC01_AC.Par.ParMonTimeMid := 0;
   A_3225_TSC01_AC.Par.ParMonTimeH := 0;
   A_3225_TSC01_AC.Par.ParMonTimeHH := 0;
   A_3225_TSC01_AC.Par.ParDelayTimeDown := 10;
   A_3225_TSC01_AC.Par.ParDelayTimeUp := 10;
   A_3225_TSC01_AC.Par.ParDelayTime := 30;
   A_3225_TSC01_AC.Par.OutMonTimeLL := 0;
   A_3225_TSC01_AC.Par.OutMonTimeL := 0;
   A_3225_TSC01_AC.Par.OutMonTimeMid := 0;
   A_3225_TSC01_AC.Par.OutMonTimeH := 0;
   A_3225_TSC01_AC.Par.OutMonTimeHH := 0;
   A_3225_TSC01_AC.Par.OutDelayTimeDown := 0;
   A_3225_TSC01_AC.Par.OutDelayTimeUp := 0;
   A_3225_TSC01_AC.Par.OutDelayTime := 0;
   A_3225_TSC01_AC.Par.Spare66 := 0;
   A_3225_TSC01_AF.StCode := 0;
   A_3225_TSC01_AF.InMonLL := FALSE;
   A_3225_TSC01_AF.InMonL := FALSE;
   A_3225_TSC01_AF.InMonMid := FALSE;
   A_3225_TSC01_AF.InMonH := FALSE;
   A_3225_TSC01_AF.InMonHH := FALSE;
   A_3225_TSC01_AF.spare0205 := FALSE;
   A_3225_TSC01_AF.InpFaultAI := FALSE;
   A_3225_TSC01_AF.InpFaultDev := FALSE;
   A_3225_TSC01_AF.InHWStop := FALSE;
   A_3225_TSC01_AF.InDPFault := FALSE;
   A_3225_TSC01_AF.InDisable := FALSE;
   A_3225_TSC01_AF.CmdFaultReset := FALSE;
   A_3225_TSC01_AF.InLocal := FALSE;
   A_3225_TSC01_AF.spare0305 := FALSE;
   A_3225_TSC01_AF.InReport := FALSE;
   A_3225_TSC01_AF.spare0307 := FALSE;
   A_3225_TSC01_AF.OutLL := FALSE;
   A_3225_TSC01_AF.OutL := FALSE;
   A_3225_TSC01_AF.OutH := FALSE;
   A_3225_TSC01_AF.OutHH := FALSE;
   A_3225_TSC01_AF.OutOverflow := FALSE;
   A_3225_TSC01_AF.spare0405 := FALSE;
   A_3225_TSC01_AF.OutFaultAI := FALSE;
   A_3225_TSC01_AF.spare0407 := FALSE;
   A_3225_TSC01_AF.StLL := FALSE;
   A_3225_TSC01_AF.StL := FALSE;
   A_3225_TSC01_AF.StMid := FALSE;
   A_3225_TSC01_AF.StH := FALSE;
   A_3225_TSC01_AF.StHH := FALSE;
   A_3225_TSC01_AF.StFaultAI := FALSE;
   A_3225_TSC01_AF.OutWarning := FALSE;
   A_3225_TSC01_AF.OutFaulted := FALSE;
   A_3225_TSC01_AF.InpValue := 0;
   A_3225_TSC01_AF.OutValuePc := 0;
   A_3225_TSC01_AF.OutValueUnits := L#0;
   A_3225_TSC01_AF.Msg.WarningDoneLL := FALSE;
   A_3225_TSC01_AF.Msg.WarningDoneL := FALSE;
   A_3225_TSC01_AF.Msg.WarningDoneMid := FALSE;
   A_3225_TSC01_AF.Msg.WarningDoneH := FALSE;
   A_3225_TSC01_AF.Msg.WarningDoneHH := FALSE;
   A_3225_TSC01_AF.Msg.FaultDoneLL := FALSE;
   A_3225_TSC01_AF.Msg.FaultDoneL := FALSE;
   A_3225_TSC01_AF.Msg.FaultDoneMid := FALSE;
   A_3225_TSC01_AF.Msg.FaultDoneH := FALSE;
   A_3225_TSC01_AF.Msg.FaultDoneHH := FALSE;
   A_3225_TSC01_AF.Msg.FaultDoneDev := FALSE;
   A_3225_TSC01_AF.Msg.FaultDoneAI := FALSE;
   A_3225_TSC01_AF.OutAlarmNrLog := 0;
   A_3225_TSC01_AF.Par.ParObjectNo := 29711;
   A_3225_TSC01_AF.Par.ParMsgType := 7252;
   A_3225_TSC01_AF.Par.ParHornCode := 11;
   A_3225_TSC01_AF.Par.ParLogOff := FALSE;
   A_3225_TSC01_AF.Par.ParSpare0401 := FALSE;
   A_3225_TSC01_AF.Par.ParValueByUser := FALSE;
   A_3225_TSC01_AF.Par.ParLimitsPc := TRUE;
   A_3225_TSC01_AF.Par.ParWago := FALSE;
   A_3225_TSC01_AF.Par.ParNoHornByWarning := FALSE;
   A_3225_TSC01_AF.Par.ParWarningLL := FALSE;
   A_3225_TSC01_AF.Par.ParWarningL := FALSE;
   A_3225_TSC01_AF.Par.ParWarningMid := FALSE;
   A_3225_TSC01_AF.Par.ParWarningH := FALSE;
   A_3225_TSC01_AF.Par.ParWarningHH := FALSE;
   A_3225_TSC01_AF.Par.ParPreAlarmLL := FALSE;
   A_3225_TSC01_AF.Par.ParPreAlarmL := FALSE;
   A_3225_TSC01_AF.Par.ParPreAlarmMid := FALSE;
   A_3225_TSC01_AF.Par.ParPreAlarmH := FALSE;
   A_3225_TSC01_AF.Par.ParPreAlarmHH := FALSE;
   A_3225_TSC01_AF.Par.ParUnitsByZeroDigit := L#0;
   A_3225_TSC01_AF.Par.ParUnitsByMaxDigit := L#16880;
   A_3225_TSC01_AF.Par.ParUnitsBy100Pc := L#10000;
   A_3225_TSC01_AF.Par.ParLimitLL := L#-1;
   A_3225_TSC01_AF.Par.ParLimitL := L#3000;
   A_3225_TSC01_AF.Par.ParLimitH := L#10000;
   A_3225_TSC01_AF.Par.ParLimitHH := L#10100;
   A_3225_TSC01_AF.Par.ParMonTimeLL := 0;
   A_3225_TSC01_AF.Par.ParMonTimeL := 0;
   A_3225_TSC01_AF.Par.ParMonTimeMid := 0;
   A_3225_TSC01_AF.Par.ParMonTimeH := 0;
   A_3225_TSC01_AF.Par.ParMonTimeHH := 0;
   A_3225_TSC01_AF.Par.ParDelayTimeDown := 10;
   A_3225_TSC01_AF.Par.ParDelayTimeUp := 10;
   A_3225_TSC01_AF.Par.ParDelayTime := 30;
   A_3225_TSC01_AF.Par.OutMonTimeLL := 0;
   A_3225_TSC01_AF.Par.OutMonTimeL := 0;
   A_3225_TSC01_AF.Par.OutMonTimeMid := 0;
   A_3225_TSC01_AF.Par.OutMonTimeH := 0;
   A_3225_TSC01_AF.Par.OutMonTimeHH := 0;
   A_3225_TSC01_AF.Par.OutDelayTimeDown := 0;
   A_3225_TSC01_AF.Par.OutDelayTimeUp := 0;
   A_3225_TSC01_AF.Par.OutDelayTime := 0;
   A_3225_TSC01_AF.Par.Spare66 := 0;
   A_3225_TSC01_AP.StCode := 0;
   A_3225_TSC01_AP.InMonLL := FALSE;
   A_3225_TSC01_AP.InMonL := FALSE;
   A_3225_TSC01_AP.InMonMid := FALSE;
   A_3225_TSC01_AP.InMonH := FALSE;
   A_3225_TSC01_AP.InMonHH := FALSE;
   A_3225_TSC01_AP.spare0205 := FALSE;
   A_3225_TSC01_AP.InpFaultAI := FALSE;
   A_3225_TSC01_AP.InpFaultDev := FALSE;
   A_3225_TSC01_AP.InHWStop := FALSE;
   A_3225_TSC01_AP.InDPFault := FALSE;
   A_3225_TSC01_AP.InDisable := FALSE;
   A_3225_TSC01_AP.CmdFaultReset := FALSE;
   A_3225_TSC01_AP.InLocal := FALSE;
   A_3225_TSC01_AP.spare0305 := FALSE;
   A_3225_TSC01_AP.InReport := FALSE;
   A_3225_TSC01_AP.spare0307 := FALSE;
   A_3225_TSC01_AP.OutLL := FALSE;
   A_3225_TSC01_AP.OutL := FALSE;
   A_3225_TSC01_AP.OutH := FALSE;
   A_3225_TSC01_AP.OutHH := FALSE;
   A_3225_TSC01_AP.OutOverflow := FALSE;
   A_3225_TSC01_AP.spare0405 := FALSE;
   A_3225_TSC01_AP.OutFaultAI := FALSE;
   A_3225_TSC01_AP.spare0407 := FALSE;
   A_3225_TSC01_AP.StLL := FALSE;
   A_3225_TSC01_AP.StL := FALSE;
   A_3225_TSC01_AP.StMid := FALSE;
   A_3225_TSC01_AP.StH := FALSE;
   A_3225_TSC01_AP.StHH := FALSE;
   A_3225_TSC01_AP.StFaultAI := FALSE;
   A_3225_TSC01_AP.OutWarning := FALSE;
   A_3225_TSC01_AP.OutFaulted := FALSE;
   A_3225_TSC01_AP.InpValue := 0;
   A_3225_TSC01_AP.OutValuePc := 0;
   A_3225_TSC01_AP.OutValueUnits := L#0;
   A_3225_TSC01_AP.Msg.WarningDoneLL := FALSE;
   A_3225_TSC01_AP.Msg.WarningDoneL := FALSE;
   A_3225_TSC01_AP.Msg.WarningDoneMid := FALSE;
   A_3225_TSC01_AP.Msg.WarningDoneH := FALSE;
   A_3225_TSC01_AP.Msg.WarningDoneHH := FALSE;
   A_3225_TSC01_AP.Msg.FaultDoneLL := FALSE;
   A_3225_TSC01_AP.Msg.FaultDoneL := FALSE;
   A_3225_TSC01_AP.Msg.FaultDoneMid := FALSE;
   A_3225_TSC01_AP.Msg.FaultDoneH := FALSE;
   A_3225_TSC01_AP.Msg.FaultDoneHH := FALSE;
   A_3225_TSC01_AP.Msg.FaultDoneDev := FALSE;
   A_3225_TSC01_AP.Msg.FaultDoneAI := FALSE;
   A_3225_TSC01_AP.OutAlarmNrLog := 0;
   A_3225_TSC01_AP.Par.ParObjectNo := 29712;
   A_3225_TSC01_AP.Par.ParMsgType := 7252;
   A_3225_TSC01_AP.Par.ParHornCode := 11;
   A_3225_TSC01_AP.Par.ParLogOff := FALSE;
   A_3225_TSC01_AP.Par.ParSpare0401 := FALSE;
   A_3225_TSC01_AP.Par.ParValueByUser := FALSE;
   A_3225_TSC01_AP.Par.ParLimitsPc := TRUE;
   A_3225_TSC01_AP.Par.ParWago := FALSE;
   A_3225_TSC01_AP.Par.ParNoHornByWarning := FALSE;
   A_3225_TSC01_AP.Par.ParWarningLL := FALSE;
   A_3225_TSC01_AP.Par.ParWarningL := FALSE;
   A_3225_TSC01_AP.Par.ParWarningMid := FALSE;
   A_3225_TSC01_AP.Par.ParWarningH := FALSE;
   A_3225_TSC01_AP.Par.ParWarningHH := FALSE;
   A_3225_TSC01_AP.Par.ParPreAlarmLL := FALSE;
   A_3225_TSC01_AP.Par.ParPreAlarmL := FALSE;
   A_3225_TSC01_AP.Par.ParPreAlarmMid := FALSE;
   A_3225_TSC01_AP.Par.ParPreAlarmH := FALSE;
   A_3225_TSC01_AP.Par.ParPreAlarmHH := FALSE;
   A_3225_TSC01_AP.Par.ParUnitsByZeroDigit := L#0;
   A_3225_TSC01_AP.Par.ParUnitsByMaxDigit := L#16384;
   A_3225_TSC01_AP.Par.ParUnitsBy100Pc := L#10000;
   A_3225_TSC01_AP.Par.ParLimitLL := L#-1;
   A_3225_TSC01_AP.Par.ParLimitL := L#0;
   A_3225_TSC01_AP.Par.ParLimitH := L#3150;
   A_3225_TSC01_AP.Par.ParLimitHH := L#3500;
   A_3225_TSC01_AP.Par.ParMonTimeLL := 0;
   A_3225_TSC01_AP.Par.ParMonTimeL := 0;
   A_3225_TSC01_AP.Par.ParMonTimeMid := 0;
   A_3225_TSC01_AP.Par.ParMonTimeH := 0;
   A_3225_TSC01_AP.Par.ParMonTimeHH := 0;
   A_3225_TSC01_AP.Par.ParDelayTimeDown := 10;
   A_3225_TSC01_AP.Par.ParDelayTimeUp := 10;
   A_3225_TSC01_AP.Par.ParDelayTime := 30;
   A_3225_TSC01_AP.Par.OutMonTimeLL := 0;
   A_3225_TSC01_AP.Par.OutMonTimeL := 0;
   A_3225_TSC01_AP.Par.OutMonTimeMid := 0;
   A_3225_TSC01_AP.Par.OutMonTimeH := 0;
   A_3225_TSC01_AP.Par.OutMonTimeHH := 0;
   A_3225_TSC01_AP.Par.OutDelayTimeDown := 0;
   A_3225_TSC01_AP.Par.OutDelayTimeUp := 0;
   A_3225_TSC01_AP.Par.OutDelayTime := 0;
   A_3225_TSC01_AP.Par.Spare66 := 0;
   A_3225_TSC01_AT.StCode := 0;
   A_3225_TSC01_AT.InMonLL := FALSE;
